//20://NG流道伺服上电
//	fbNGStepMotor.xPowerInit:=TRUE;
//	IF     fbNGStepMotor.xPowerOn THEN
//		station.iStepInit :=30;
//	END_IF
30://判断电动夹爪是否可以初始化
	IF    (tsModuleProcess[4].xProcessStarted AND  NOT tsModuleProcess[4].xProcessCompleted) OR
		  (tsModuleProcess[5].xProcessStarted AND  NOT tsModuleProcess[5].xProcessCompleted)  OR test THEN
			station.iStepInit :=50;(*电动夹爪不能初始h化*)
	ELSE
			station.iStepInit :=40;
	END_IF
40://大寰夹爪初始化
		fbClamp.stOper.xInitControl:=TRUE ;	
		 IF fbClamp.xDone  THEN 
				fbClamp.xExecute :=FALSE;
				station.iStepInit:=45;
		 END_IF	
45://大寰夹爪张开
			fbClamp.stOper.aReleaseControl[1]:=TRUE ;
				IF fbClamp.xDone  THEN 
					fbClamp.xExecute :=FALSE ;
					station.iStepInit:= 50;
				END_IF		
50:  //机械手初始化
		stToRobot1.iMoveMode := CmdRobot1.Cmd_GoHome ;//切换到回原点
		fbRobot.xInitExte := TRUE ;	
		station.iStepInit:=60;		
60:
		IF fbRobot.xInitFinish THEN 
			fbRobot.xInitExte := FALSE ;	
			station.iStepInit:=65;		
		END_IF		
65:
			//stToRobot1.iMoveMode := CmdRobot1.Cmd_GoHome ;
			station.iStepInit:=70;	
70://机械手初始化	
		IF  stFromRobot1.xStepRunning THEN
		 		station.iStepInit:=80;	
				stToRobot1.iMoveMode := CmdRobot1.noCmd ;
		END_IF
80://运行初始化子程序
		stToRobot1.xStepRunPermit := TRUE ;
	 IF stFromRobot1.xStepRunDone  THEN
		stToRobot1.xStepRunPermit := FALSE ;
   		station.iStepInit:=90;	
	 END_IF
90://机械手初始化并检测机械手初始化完成
	 IF  stFromRobot1.xHomePosReached THEN
        station.iStepInit:=999;	
	 END_IF	

999://初始化完成	
	station.iStepInit:=0;
	station.xInitDone:=TRUE;  
END_CASE
END_IF
END_ACTION

ACTION General:
EstopR_TRIG(CLK:= NOT  fbMachine[1].xEStop , Q=> );
IF  EstopR_TRIG.Q THEN 
		xS07MainlineRunPermit:=FALSE;
END_IF
MachineInitR_TRIG(CLK:=fbMachine[1].xIniting , Q=> );
IF MachineInitR_TRIG.Q THEN
		bRobCounter :=0;
END_IF
END_ACTION

ACTION ILC:

//---------------------------------------------------工站可执行-------------------------------------------------------
station.xCanRun :=TRUE ;

//---------------------------------------------------伺服动作条件-------------------------------------------
fbNGStepMotor.xRunILC := TRUE;
fbNGStepMotor.xMoveILC[1] :=TRUE;
//大寰夹爪
fbClamp.xDeviceRunning:=station.xSingleRunning OR   station.xIniting OR   station.xRunning ;
END_ACTION

ACTION TipAuto:

//------------------------------------------------AutoTip Cylinder--------------------------------

//------------------------------------------------AutoTip Servo--------------------------------
//**************************************
//FOR i:= 1 TO 5 BY 1 DO 
//	IF fbNGStepMotor.xMoveAuto[i] THEN
//		fbNGStepMotor.iPosNumber := i ;
//	END_IF
//	
//END_FOR
//
//
//IF  fbMachine[1].xAutoMode AND NOT fbMachine[1].xRunning AND  arTonDelay[10].Q   THEN
//		IF	fbNGStepMotor.iPosNumber=1 	AND NOT fbNGStepMotor.xMoveInPos[1] THEN 	station.adwAutoTip[1].10:=TRUE	;	END_IF//轴伺服自动时位置不在位置1
//		IF	fbNGStepMotor.iPosNumber=2	AND NOT fbNGStepMotor.xMoveInPos[2]	THEN 	station.adwAutoTip[1].11:=TRUE	;	END_IF//轴伺服自动时位置不在位置2
//		IF	fbNGStepMotor.iPosNumber=3	AND NOT fbNGStepMotor.xMoveInPos[3]	THEN 	station.adwAutoTip[1].12:=TRUE	;	END_IF//轴伺服自动时位置不在位置3
//		IF	fbNGStepMotor.iPosNumber=4	AND NOT fbNGStepMotor.xMoveInPos[4]	THEN 	station.adwAutoTip[1].13:=TRUE	;	END_IF//轴伺服自动时位置不在位置4
//		IF	fbNGStepMotor.iPosNumber=5	AND NOT fbNGStepMotor.xMoveInPos[5]	THEN 	station.adwAutoTip[1].14:=TRUE	;	END_IF//轴伺服自动时位置不在位置5
//END_IF
//
END_ACTION

ACTION TipManual:
//--------------------------------------------ManualTip------------------------------------------------------

//-------------------------------------------气缸提示---------------------------------------------------------




/////////////////////////////////////////////////////////////////////////////////////////////////////////////////
END_ACTION

ACTION Z_Output:
(*
CASE  bRobotStep  OF
 0:
 		IF   xRobotStartTryRun  THEN
		 		 bRobotStep:=bRobotStep +1;
		END_IF
1:  //机械手初始化
		fbRobot.xInitExte := TRUE ;
		 bRobotStep:=bRobotStep +1;
2:
		IF fbRobot.xInitFinish THEN 
			fbRobot.xInitExte := FALSE ;	
			 bRobotStep:=bRobotStep +1;
		END_IF		
3://机械手初始化	
		stToRobot1.iMoveMode := CmdRobot1.Cmd_GoHome ;
		IF  stFromRobot1.xStepRunning THEN
		 		 bRobotStep:=bRobotStep +1;
				stToRobot1.iMoveMode := CmdRobot1.noCmd ;
		END_IF
4://运行初始化子程序
		stToRobot1.xStepRunPermit := TRUE ;
	 IF stFromRobot1.xStepRunDone  THEN
		stToRobot1.xStepRunPermit := FALSE ;
   	 bRobotStep:=bRobotStep +1;
	 END_IF
5://机械手初始化并检测机械手初始化完成
	 IF  stFromRobot1.xHomePosReached THEN
       bRobotStep:=bRobotStep +1;
	 END_IF	
6://机械手选择取料程序	
			stToRobot1.iMoveMode := CmdRobot1.Cmd_TakePart ;//切换程序
			IF    stFromRobot1.xStepRunning  THEN
			 			stToRobot1.iMoveMode := CmdRobot1.noCmd ;
			 			 bRobotStep:=bRobotStep +1;
			END_IF
7://取料子程序运行
			stToRobot1.xStepRunPermit := TRUE ;
			IF stFromRobot1.xStepRunDone THEN
					stToRobot1.xStepRunPermit := FALSE ;
					 bRobotStep:=bRobotStep +1;
	 		END_IF
8:	//机械手允许去取料位
				 	stToRobot1.xPickPos1Premit :=TRUE;
						IF stFromRobot1.xPickPos1Reached THEN 
							 stToRobot1.xPickPos1Premit := FALSE ;
							 	 bRobotStep:=bRobotStep +1;
						END_IF
9://夹取完成,机械手回中转位
				stToRobot1.xClampPartDone:=TRUE;
			IF   stFromRobot1.xPickTransferPosReached THEN
					 bRobotStep:=bRobotStep +1;
			END_IF
10:
			stToRobot1.iMoveMode := CmdRobot1.Cmd_PutPart ;//切换程序
			IF    stFromRobot1.xStepRunning  THEN
			 			stToRobot1.iMoveMode := CmdRobot1.noCmd ;
			 		 bRobotStep:=bRobotStep +1;
			END_IF
11://放料子程序运行
			stToRobot1.xStepRunPermit := TRUE ;
			IF stFromRobot1.xStepRunDone THEN
					stToRobot1.xStepRunPermit := FALSE ;
					 bRobotStep:=bRobotStep +1;
	 		END_IF
12:	//机械手开始放料
			stToRobot1.xPutPos1Premit:=TRUE;(*卡片1位置 *)
			IF stFromRobot1.xPutPos1Reached THEN 
				 stToRobot1.xPutPos1Premit := FALSE ;
				 bRobotStep:=bRobotStep +1;
			END_IF
13://机械手回中转位置
			stToRobot1.xReleasePartDone:=TRUE;
			IF stFromRobot1.xPickTransferPosReached THEN
					bRobotStep:=0;
	 		END_IF	
END_CASE
*)
END_ACTION

END_PROGRAM

// ---- POUs/003_FB/0013_RGI_14_new/不带旋转的电动夹爪/FB_RGI_14_Modbus.TcPOU
{attribute 'tc_no_symbol'}
FUNCTION_BLOCK FB_RGI_14_Modbus
VAR_INPUT
	xExecute: BOOL;
	xAbort: BOOL;
	xPowerHmi: BOOL := TRUE;
	////上电信号，反转型
	xResetRequest: BOOL;
	///[ms],1 => no invocation time limit
	dwTimeLimit: DWORD := 1;
	///[ms],0 => no executing time limit 
	dwTimeOut: DWORD;
	///系统参数
	stPara: ST_RGI_14_Sys_Para;
	///0:mannal 1:auto
	xAutoMode: BOOL;
	///初始化过程中	
	xIniting: BOOL;
	///参数设置
	stPosPara: ST_RGI_PosPara;
	///流程运行过程中
	xDeviceRunning: BOOL;
	///手动自动操作
	stOper: ST_RGI_Opera;
END_VAR
VAR_OUTPUT
	///完成条件满足
	xDone: BOOL;
	///动作正在执行
	xBusy: BOOL;
	///指令被打断
	xAborted: BOOL;
	///错误条件满足
	xError: BOOL;
	///错误码
	eErrorID: RGI_14_ERROR;
	///eMobbusErrorID: MODBUS_ERROR;//modubs 报警信息
	xRdyCmd: BOOL;
	xRefOk: BOOL;
	eClampActCmd: RGI_14_CMD;
	///0：运动中，1：到达位置；2：夹住物体；3：物体掉落	
	iClampStatus: INT;
	///夹爪夹空
	xGripClampEmpty: BOOL;
	///掉落发生
	xDropOccur: BOOL;
	///关盖失败
	xClosecoverFailure: BOOL;
	///开盖失败
	xOpencoverFailure: BOOL;
	sHmiError: STRING;
	stRGIStates: ST_RGI_HMIStates;
	eCommErrorID: BYTE;
	eOperErrorID: DWORD;
END_VAR
VAR_IN_OUT
	st_IOData: ST_RGI_14_IOData;
END_VAR
VAR
	{attribute 'tc_no_symbol'}
	_xDone: BOOL;
	{attribute 'tc_no_symbol'}
	eCmd: RGI_14_CMD;
	{attribute 'tc_no_symbol'}
	///目标力值设置
	iTorqueSet: INT := 50;
	{attribute 'tc_no_symbol'}
	///运行速度设置
	iSpeedSet: INT := 50;
	{attribute 'tc_no_symbol'}
	///位置和速度设置值	
	iPosAngleSet: INT := 500;
	{attribute 'tc_no_symbol'}
	eState: STATE;
	{attribute 'tc_no_symbol'}
	xFirstInvocation: BOOL := TRUE;
	{attribute 'tc_no_symbol'}
	xTimeOut: BOOL;
	{attribute 'tc_no_symbol'}
	tOperationTimer: TON;
	{attribute 'tc_no_symbol'}
	_tonTimeout: TON;
	{attribute 'tc_no_symbol'}
	_tonCmdTimeout: TON;
	{attribute 'tc_no_symbol'}
	_tonPulse: TON;
	{attribute 'tc_no_symbol'}
	_tonDelay: TON;
	{attribute 'tc_no_symbol'}
	_tonConnectDelay: TON;
	{attribute 'tc_no_symbol'}
	_tonConnectTimeout: TON;
	{attribute 'tc_no_symbol'}
	/// detect rising edge of command execution 
	_diCmdState: DINT;
	{attribute 'tc_no_symbol'}
	i: INT;
	{attribute 'tc_no_symbol'}
	ii: INT;
	{attribute 'tc_no_symbol'}
	_idx: INT;
	{attribute 'tc_no_symbol'}
	_xConnectError: BOOL;
	{attribute 'tc_no_symbol'}
	_fResetCheck: F_TRIG;
	{attribute 'tc_no_symbol'}
	_iRotateAngleLTemp: INT;
	{attribute 'tc_no_symbol'}
	_iRotateAngleHTemp: INT;
	{attribute 'tc_no_symbol'}
	_iRotateAngleTotalTemp: DINT;
	{attribute 'tc_no_symbol'}
	_iRotateAngleCurrentTemp: DINT;
	{attribute 'tc_no_symbol'}
	_xRotateFinish: BOOL;
	{attribute 'tc_no_symbol'}
	_iConnectState: INT := 0;
	{attribute 'tc_no_symbol'}
	_connectTon: TON;
	{attribute 'tc_no_symbol'}
	_rManual: R_TRIG;
	{attribute 'tc_no_symbol'}
	_fManual: F_TRIG;
	{attribute 'tc_no_symbol'}
	_xModeChange: BOOL;
	{attribute 'tc_no_symbol'}
	///上电是默认读取模式的
	_xReadStatus: BOOL := TRUE;
	{attribute 'tc_no_symbol'}
	_iCount: INT := 0;
	{attribute 'tc_no_symbol'}
	_iAbortState: INT := 0;
	{attribute 'tc_no_symbol'}
	_fPowerOn :F_TRIG;
  {attribute 'tc_no_symbol'}
	_rHMIControl: R_TRIG;
	{attribute 'tc_no_symbol'}
	_iNGCount: INT;
	{attribute 'tc_no_symbol'}
	///4:控制反馈数据，5:状态反馈数据
	_aRead_VAR: ARRAY[4..5] OF FB_MBReadRegs;
	{attribute 'tc_no_symbol'}
	///0:初始化控制；1:夹紧控制；2:旋转绝对控制；3:旋转相对控制
	_aWtirt_VAR: ARRAY[0..3] OF FB_MBWriteRegs;
	{attribute 'tc_no_symbol'}
	///0:初始化控制；1:夹紧控制；2:旋转绝对控制；3:旋转相对控制；4:控制反馈数据，5:状态反馈数据	
	_aEnableSignal: ARRAY[0..5] OF BOOL;
	{attribute 'tc_no_symbol'}
	///反馈数据	
	_aFeedbackData: ARRAY[4..5, 0..11] OF INT;
	{attribute 'tc_no_symbol'}
	///控制参数	
	_aControlData: ARRAY[0..3, 0..3] OF INT;
	{attribute 'tc_no_symbol'}
	_iChannelIndex: INT;
	{attribute 'tc_no_symbol'}
	_xConnect_ERROR: BOOL;
	{attribute 'tc_no_symbol'}
	iCMDNGIndex: INT;
	{attribute 'tc_no_symbol'}
	_xBusy: BOOL;
	{attribute 'tc_no_symbol'}
	///发送状态标志位
	_iSendReceiveState: INT := 0;
	{attribute 'tc_no_symbol'}
	_tonDelay1: TON;
	{attribute 'tc_no_symbol'}
	_tonDelay2: TON;
	{attribute 'tc_no_symbol'}
	_iComNGCount: INT;
	{attribute 'tc_no_symbol'}
	///初始化指令触发
	_rHMIInit: R_TRIG;
	{attribute 'tc_no_symbol'}
	///初始化指令触发
	_rInit: R_TRIG;
	{attribute 'tc_no_symbol'}
	///夹紧轴指令触发
	_rHMIClamp: ARRAY[1..10] OF R_TRIG;
	{attribute 'tc_no_symbol'}
	///夹紧轴指令触发
	_rHMIRelease: ARRAY[1..10] OF R_TRIG;
	{attribute 'tc_no_symbol'}
	///夹紧轴指令触发
	_rClamp: ARRAY[1..10] OF R_TRIG;
	{attribute 'tc_no_symbol'}
	///夹紧轴指令触发
	_rRelease: ARRAY[1..10] OF R_TRIG;
	{attribute 'tc_no_symbol'}
	///旋转轴指令触发	
	_rHMIRotateClamp: ARRAY[1..10] OF R_TRIG;
	{attribute 'tc_no_symbol'}
	///旋转轴指令触发	
	_rHMIRotateClampRef: ARRAY[1..10] OF R_TRIG;
	{attribute 'tc_no_symbol'}
	///旋转轴指令触发	
	_rHMIRotateRelease: ARRAY[1..10] OF R_TRIG;
	{attribute 'tc_no_symbol'}
	///旋转轴指令触发	
	_rHMIRotateReleaseRef: ARRAY[1..10] OF R_TRIG;
	{attribute 'tc_no_symbol'}
	///旋转轴指令触发	
	_rRotateClamp: ARRAY[1..10] OF R_TRIG;
	{attribute 'tc_no_symbol'}
	///旋转轴指令触发	
	_rRotateRelease: ARRAY[1..10] OF R_TRIG;
	{attribute 'tc_no_symbol'}
	///旋转轴指令触发	
	_rRotateClampRef: ARRAY[1..10] OF R_TRIG;
	{attribute 'tc_no_symbol'}
	///旋转轴指令触发	
	_rRotateReleaseRef: ARRAY[1..10] OF R_TRIG;
	{attribute 'tc_no_symbol'}
	_Angle_rec: INT;
	{attribute 'tc_no_symbol'}
	///是否有手动操作，是否有自动操作
	_xHMIOpe: BOOL;
	{attribute 'tc_no_symbol'}
	///是否有手动操作，是否有自动操作
	_xAutoOpe: BOOL;
END_VAR
VAR_TEMP
	{attribute 'tc_no_symbol'}
	xAgain: BOOL;
END_VAR

xAgain:=0;
ACTMap();//数据映射
ConnectAction();//触发通信连接功能连接
_fResetCheck(CLK:=xResetRequest OR stOper.xHMIReset);//reset
IF eState<>STATE.DORMANT
THEN
	_rHMIInit(CLK:=FALSE) ;
	_rInit(CLK:=FALSE) ;
	 FOR ii :=1 TO 10 DO
		 _rHMIClamp[ii](CLK:=FALSE);
		 _rHMIRelease[ii](CLK:=FALSE);
		 _rClamp[ii](CLK:=FALSE);
		 _rRelease[ii](CLK:=FALSE);
		 _rHMIRotateClamp[ii](CLK:=FALSE);
		 _rHMIRotateRelease[ii](CLK:=FALSE);
		 _rRotateClamp[ii](CLK:=FALSE);
		 _rRotateRelease[ii](CLK:=FALSE);
		 _rRotateClampRef[ii](CLK:=FALSE);
		 _rRotateReleaseRef[ii](CLK:=FALSE);
		 _rHMIRotateClampRef[ii](CLK:=FALSE);
		 _rHMIRotateReleaseRef[ii](CLK:=FALSE);		 
	 END_FOR
END_IF
REPEAT
	CASE eState OF
		STATE.DORMANT:
				HandleDormantState(xAgain=> xAgain);
		STATE.EXECUTING:
				HandleExecutingState(xAgain=> xAgain);
		STATE.DONE:
				HandleDoneState(xAgain=> xAgain);
		STATE.INERROR:
				HandleErrorState(xAgain=> xAgain);
		STATE.ABORTING:
				HandleAbortingState(xAgain=> xAgain);
		STATE.ABORTED:
				HandleAbortedState(xAgain=> xAgain);
		STATE.RESETING:
				HandleResettingState(xAgain=> xAgain);
	END_CASE
UNTIL (xAgain=0)
END_REPEAT

//报错信息提示	
CASE eErrorID OF
	RGI_14_ERROR.NO_ERROR:
		sHmiError:='NO_ERROR';	
  RGI_14_ERROR.FLT_PARA:
		sHmiError:='FLT_PARA';	
  RGI_14_ERROR.FLT_CONNECT:
		sHmiError:='FLT_CONNECT';	
  RGI_14_ERROR.FLT_RDYCMD:
		sHmiError:='FLT_RDYCMD';	
	RGI_14_ERROR.FLT_DEVICE_ERROR:
		sHmiError:='FLT_DEVICE_ERROR';	
	RGI_14_ERROR.FLT_POWERON:
		sHmiError:='FLT_POWERON';	
  RGI_14_ERROR.FLT_CLAMP_TIMEOUT:
		sHmiError:='FLT_CLAMP_TIMEOUT';	
  RGI_14_ERROR.FLT_ROTATE_TIMEOUT:
		sHmiError:='FLT_ROTATE_TIMEOUT';	
  RGI_14_ERROR.FLT_ORG_TIMEOUT:
		sHmiError:='FLT_ORG_TIMEOUT';	
	RGI_14_ERROR.FLT_CLAMPCMD_TIMEOUT:
		sHmiError:='FLT_CLAMPCMD_TIMEOUT';	
  RGI_14_ERROR.FLT_ROTATECMDABS_TIMEOUT:
		sHmiError:='FLT_ROTATECMDABS_TIMEOUT';
  RGI_14_ERROR.FLT_ROTATECMDREF_TIMEOUT:
		sHmiError:='FLT_ROTATECMDREF_TIMEOUT';			
  RGI_14_ERROR.FLT_ORGCMD_TIMEOUT:
		sHmiError:='FLT_ORGCMD_TIMEOUT';	
	RGI_14_ERROR.FLT_CLAMP_DROP:
		sHmiError:='FLT_CLAMP_DROP';	  
  RGI_14_ERROR.FLT_xRefOk:
		sHmiError:='FLT_xRefOk';	
	RGI_14_ERROR.FLT_CLAMP_PARA:
		sHmiError:='FLT_CLAMP_PARA';		
	RGI_14_ERROR.FLT_ClAMP_RELEASEFAIL:
		sHmiError:='FLT_ClAMP_RELEASEFAIL';	
  RGI_14_ERROR.FLT_ClAMP_CLAMPFAIL:
		sHmiError:='FLT_ClAMP_CLAMPFAIL';	
	RGI_14_ERROR.FLT_ROTATE_CLAMPFAIL:
		sHmiError:='FLT_ROTATE_CLAMPFAIL';	
	RGI_14_ERROR.FLT_ROTATE_RELEASEFAIL:
		sHmiError:='FLT_ROTATE_RELEASEFAIL';		
END_CASE

//检测是否有手动操作
_xHMIOpe := stOper.xHMInitButton;
FOR i := 1 TO 10 BY 1
DO
	_xHMIOpe := _xHMIOpe OR stOper.aHMIClampButton[i] OR stOper.aHMIReleaseButton[i] OR stOper.aHMIRotateClampButton[i] OR stOper.aHMIRotateClampRefButton[i] 
							OR stOper.aHMIRotateReleaseButton[i] OR stOper.aHMIRotateReleaseRefButton[i];
END_FOR

//检测是否有自动操作指令
_xAutoOpe := stOper.xInitControl;
FOR i := 1 TO 10 BY 1
DO
	_xAutoOpe := _xAutoOpe OR stOper.aClampControl[i] OR stOper.aReleaseControl[i] OR stOper.aRotateClampControl[i] OR stOper.aRotateClampRefControl[i] 
							OR stOper.aRotateReleaseControl[i] OR stOper.aRotateReleaseRefControl[i];
END_FOR

///{attribute 'tc_no_symbol'}
METHOD PROTECTED AbortAction
VAR_OUTPUT
	xComplete: BOOL;
	eErrorID: RGI_14_ERROR;
END_VAR
(*
* Cleaning
* => abort all running operation
* => if an NBS.ERROR codition is reached, set eErrorID to a Value rather then NBS.RGI_14_ERROR.NO_ERROR 
*)
CASE _iAbortState OF 
	0://复位所以的控制信号

	ELSE
		;	
END_CASE
END_METHOD

ACTION ACTCheckRotateFinish:
(******************************检测旋转是否完成*************************************)
_xRotateFinish := FALSE;
IF eCmd = RGI_14_CMD.Cmd_RotateAbsClamp OR eCmd = RGI_14_CMD.Cmd_RotateAbsRelease //绝对旋转模式
THEN
	//检测是否已经处于目标位置
	IF iPosAngleSet = st_IOData.I_RotateAngleL
	THEN
		_xRotateFinish := TRUE;
	END_IF	
END_IF
IF eCmd = RGI_14_CMD.Cmd_RoratRelClamp OR eCmd = RGI_14_CMD.Cmd_RoratRelRelease//增量旋转模式
THEN	
	//使用计算公式来进行预测是否已经到目标位置
	_iRotateAngleTotalTemp := _iRotateAngleHTemp * 32768 + _iRotateAngleLTemp + iPosAngleSet;
	_iRotateAngleCurrentTemp := st_IOData.I_RotateAngleH * 32768 + st_IOData.I_RotateAngleL;
	IF _iRotateAngleTotalTemp = _iRotateAngleCurrentTemp
	THEN
		_xRotateFinish := TRUE;
	END_IF
END_IF
END_ACTION

ACTION ACTMap:
//进行数据映射的前提条件是外部所配置的参数是没有问题的
IF stPara.strSlaveIP <> '' 
THEN
	//夹爪设置反馈
	st_IOData.i_Init			:=_aFeedbackData[4,0];
	st_IOData.i_ClampForceSet	:=_aFeedbackData[4,1];
	
	st_IOData.i_ClampPosSet		:=_aFeedbackData[4,3];	
	st_IOData.i_ClampSpeedSet	:=_aFeedbackData[4,4];
	st_IOData.i_RotateAngleLSet	:=_aFeedbackData[4,5];
	st_IOData.i_RotateAngleHSet	:=_aFeedbackData[4,6];
	st_IOData.i_RotateSpeedSet	:=_aFeedbackData[4,7];
	st_IOData.i_RotateForseSet	:=_aFeedbackData[4,8];
	st_IOData.i_RotateRelAngle	:=_aFeedbackData[4,9];
	
	//夹爪状态反馈
	st_IOData.I_ClampInit := _aFeedbackData[5,0];
	st_IOData.I_ClampState := _aFeedbackData[5,1];
	st_IOData.I_CurrentPos := _aFeedbackData[5,2];
	st_IOData.I_DeviceERRORState := _aFeedbackData[5,5];
	st_IOData.I_RotateAngleL := _aFeedbackData[5,8];
	st_IOData.I_RotateAngleH := _aFeedbackData[5,9];
	st_IOData.I_RotateInit := _aFeedbackData[5,10];
	st_IOData.I_RotateState := _aFeedbackData[5,11];			
	//夹爪状态
	iClampStatus := st_IOData.I_ClampState ;
	
	//进行输出数据刷新(外面一定要用保持性的数据来定义)
	_aControlData[0,0] := st_IOData.O_Init;//同时初始化夹紧轴和旋转轴
	_aControlData[1,0] := st_IOData.O_ClampForceSet;//夹紧力值设计
	_aControlData[1,2] := st_IOData.O_ClampPosSet;//夹紧位置设置
	_aControlData[1,3] := st_IOData.O_ClampSpeedSet;//夹紧速度设置
	//旋转绝对定位
	IF eCmd = RGI_14_CMD.Cmd_RotateAbsClamp OR eCmd = RGI_14_CMD.Cmd_RotateAbsRelease
	THEN
		_aControlData[2,0]	:= st_IOData.O_RotateAngleLSet;//绝对旋转角度设置1
		_aControlData[2,1] := st_IOData.O_RotateAngleHSet;//绝对旋转角度设置2	
		_aControlData[2,2] := st_IOData.O_RotateSpeedSet;//旋转速度设计
		_aControlData[2,3] := st_IOData.O_RotateForseSet;//旋转力值设计		
	END_IF
	//旋转相对定位
	IF eCmd = RGI_14_CMD.Cmd_RoratRelClamp OR eCmd = RGI_14_CMD.Cmd_RoratRelRelease
	THEN
		_aControlData[3,0] := st_IOData.O_RotateSpeedSet;//旋转速度设计
		_aControlData[3,1] := st_IOData.O_RotateForseSet;//旋转力值设计
		_aControlData[3,2] := st_IOData.O_RotateRelAngle;//旋转相对角度设计
	END_IF
	
END_IF

(****************************夹紧轴状态读取(此时一定是模块连接上的，此时刷新周期不要太短，兼容效率***************************)
_tonPulse(IN:=NOT _tonPulse.Q , PT:=T#200MS);//产生100ms的脉冲信号
IF _xReadStatus  //一定要处于通信正常状态
THEN
	_aRead_VAR[5].bExecute := _tonPulse.Q;//保证通信不断
END_IF

xRdyCmd := xPowerHmi AND(( eState = STATE.DORMANT ) OR (NOT xAutoMode AND _xAutoOpe AND eState = STATE.DONE ));//rdy显示变化;
_rInit(CLK:= xIniting);//检测是否是初始化中，如果是的去切换模式
IF _rInit.Q
THEN
 eState := STATE.RESETING;
END_IF 
//检测是否有模式变化
_fManual(CLK:=xAutoMode);
_rManual(CLK:=xAutoMode);
IF eState <> STATE.DORMANT//只有在运行的时候，才会检测是否有模式切换发生
THEN
	IF _fManual.Q OR _rManual.Q
	THEN
		_xModeChange := TRUE;
	END_IF
END_IF

(****************************电源控制********************************************)

_fPowerOn(CLK:= xPowerHmi);//驱动器断电的时候需要将初始化完成信号给清除掉
IF _fPowerOn.Q
THEN
	xRefOk := FALSE;//断电再上电之后需要重新初始化
END_IF

(*****************************夹爪状态显示*****************************)
xDone := _xDone AND xExecute;//判断是否处于当前流程的Done状态
xDropOccur :=( eClampActCmd = RGI_14_CMD.Cmd_Clamp ) AND ( st_IOData.I_ClampState = 3 );
xGripClampEmpty := xError AND eErrorID = RGI_14_ERROR.FLT_ClAMP_CLAMPFAIL AND xExecute;//关盖失败判定
xClosecoverFailure := xError AND eErrorID = RGI_14_ERROR.FLT_ROTATE_CLAMPFAIL AND xExecute;//关盖失败判定
xOpencoverFailure := xError AND eErrorID = RGI_14_ERROR.FLT_ROTATE_RELEASEFAIL AND xExecute;//开盖失败评定

(*****************************触摸屏状态显示*****************************)
stRGIStates.xDone:=xDone;
stRGIStates.xBusy:=xBusy;
stRGIStates.xRefOk:=xRefOk;
stRGIStates.xRdyCmd:=xRdyCmd;
stRGIStates.eErrorID:=eErrorID;
stRGIStates.sHmiError:=sHmiError;
stRGIStates.iClampStatus:=iClampStatus;
stRGIStates.xClosecoverFailure:=xClosecoverFailure;
stRGIStates.xGripClampEmpty:=xGripClampEmpty;
stRGIStates.xOpencoverFailure:=xOpencoverFailure;
stRGIStates.xGripClampEmpty:=xGripClampEmpty;
stRGIStates.xError:=xError;
END_ACTION

METHOD PROTECTED CmdClampAction
VAR_OUTPUT
	xComplete: BOOL;
END_VAR
// return the real actual fault number
IF eErrorID <> RGI_14_ERROR.NO_ERROR
THEN
  RETURN;  
END_IF
  
IF NOT xRefOk THEN
	eErrorID := RGI_14_ERROR.FLT_xRefOk;
	RETURN;
END_IF

IF iPosAngleSet < 0 OR iPosAngleSet > 1000//夹紧参数错误
THEN
	eErrorID := RGI_14_ERROR.FLT_CLAMP_PARA;
	RETURN;
END_IF

CASE _diCmdState OF
	0://判断对应指令，是否已经处于完成状态，防止出现重复触发情况
		_tonDelay(IN:= FALSE);
		IF NOT _aRead_VAR[5].bExecute THEN		
			_diCmdState := _diCmdState + 1;
		END_IF	
		
	1://传送力值和速度参数
		_tonDelay(IN:= TRUE,pt:=T#20MS);
		st_IOData.O_ClampForceSet	:= iTorqueSet;
		st_IOData.O_ClampSpeedSet	:= iSpeedSet;	
		st_IOData.O_ClampPosSet 	:= iPosAngleSet;	
		IF _tonDelay.Q 
		THEN
			//复位定时器
				_tonDelay(IN:=FALSE);
				_tonCmdTimeout(in:=FALSE);
				_tonTimeout(in:=FALSE);	
			 _aEnableSignal[1]:=TRUE;	
			 _diCmdState := _diCmdState+1;
	 END_IF				
		
	2://等待反应，设置读取参数
		_tonDelay(IN:= NOT _aEnableSignal[1],PT:=T#300MS);//此时电动夹爪一定已经响应
		IF _tonDelay.Q//
		THEN		
			_diCmdState := _diCmdState +1;			
		END_IF	
		
		IF _iSendReceiveState = 999
		THEN
			iCMDNGIndex := 1;
			eErrorID := RGI_14_ERROR.FLT_CLAMPCMD_TIMEOUT;		
			_diCmdState := 999;
		END_IF	
		
	3://读取数据
		_tonCmdTimeout(in:=FALSE);
		_tonDelay(IN:=FALSE);	
		_tonTimeout(in:=TRUE,pt:=T#10S);//设置超时时间 
		_aEnableSignal[5] := TRUE;//触发读取反馈数据	
		_diCmdState := _diCmdState +1; 
	
	4://等待运行完成
		_tonTimeout(in:=TRUE,pt:=T#10S); 
		_tonCmdTimeout(IN:= TRUE,pt:=T#2S);				
		IF NOT _aEnableSignal[5] //等待读取数据完成
		THEN	
			_tonDelay(IN:= TRUE,pt:=T#40MS);//设置刷新周期
			IF _tonDelay.Q
			THEN
				_diCmdState := 3;//回到上一步重新进行状态刷新
			END_IF
			
			IF (st_IOData.I_ClampState = 1 OR stOper.xTestMode )AND st_IOData.O_ClampPosSet = st_IOData.I_CurrentPos AND //松开位置成功
			   eCmd = RGI_14_CMD.Cmd_Release	//松开指令
			THEN			
				_tonCmdTimeout(in:=FALSE);
				_tonTimeout(in:=FALSE);  
				_diCmdState := 100;
				xComplete := TRUE;
			END_IF		
			IF (st_IOData.I_ClampState = 2 OR stOper.xTestMode) AND//夹住物体
				 eCmd = RGI_14_CMD.Cmd_Clamp	//夹紧指令
			THEN			
				_tonTimeout(in:=FALSE);  
				_diCmdState := 100;
				xComplete := TRUE;
			END_IF			
		//非测试模式才启动检测
		IF NOT stOper.xTestMode THEN	
			IF st_IOData.I_ClampState = 2 AND //松开位置的时候，没有松开到位置，松开失败
				 eCmd = RGI_14_CMD.Cmd_Release	//松开指令
			THEN	
				_iNGCount := _iNGCount + 1;		
				IF _iNGCount <= 3
				THEN
					_tonDelay(IN:=FALSE);
					_diCmdState := _diCmdState + 1;
				ELSE
					_tonTimeout(in:=FALSE);  
					eErrorID := RGI_14_ERROR.FLT_ClAMP_RELEASEFAIL;		
					_diCmdState := 999;
				END_IF				
			END_IF		
			IF st_IOData.I_ClampState = 1 AND st_IOData.O_ClampPosSet = st_IOData.I_CurrentPos AND//没有夹住物体，到位置，判定夹持失败
				 eCmd = RGI_14_CMD.Cmd_Clamp	//夹紧指令
			THEN
				_iNGCount := _iNGCount + 1;		
				IF _iNGCount <= 3
				THEN
					_tonDelay(IN:=FALSE);
					_diCmdState := _diCmdState + 1;
				ELSE
					_tonCmdTimeout(in:=FALSE);
					_tonTimeout(in:=FALSE);  			
					eErrorID := RGI_14_ERROR.FLT_ClAMP_CLAMPFAIL;		
					_diCmdState := 999;
				END_IF
			END_IF		
		END_IF
	END_IF
	
	IF _iSendReceiveState = 999//旋转指令响应超时
	THEN
		iCMDNGIndex := 3;
		eErrorID := RGI_14_ERROR.FLT_CLAMPCMD_TIMEOUT;		
		_diCmdState := 999;
	END_IF		
	
	IF _tonTimeout.Q//旋转动作超时
	THEN
		_iNGCount := _iNGCount + 1;
		IF _iNGCount >= 2
		THEN
			eErrorID := RGI_14_ERROR.FLT_CLAMP_TIMEOUT;
			_diCmdState := 999;
		ELSE
			_aEnableSignal[5] := FALSE;
			_diCmdState := 0;
		END_IF
	END_IF
	
	5://报警再次确定
		_tonDelay(IN:= TRUE,pt:=T#50MS);
		IF _tonDelay.Q//做延时刷新
		THEN			
			_diCmdState :=3;
		END_IF
			
ELSE
	;	
END_CASE
END_METHOD

METHOD PROTECTED CmdRotateAction_ABS
VAR_OUTPUT
	xComplete: BOOL;
END_VAR
// return the real actual fault number
IF eErrorID <> RGI_14_ERROR.NO_ERROR
THEN
  RETURN;  
END_IF
  
IF NOT xRefOk THEN//设备没有原点报警
	eErrorID := RGI_14_ERROR.FLT_xRefOk;
	RETURN;
END_IF

CASE _diCmdState OF
	0://判断是否已经处于目标位置或者夹取完成状态，防止出现重复触发情况
		_tonDelay(IN:= FALSE);
		IF NOT _aRead_VAR[5].bExecute THEN		
			_diCmdState := _diCmdState + 1;
		END_IF		
		
	1://传送参数	
		_tonDelay(IN:= TRUE,PT:=T#20MS);//等待设备运行起来
		_iRotateAngleLTemp := st_IOData.I_RotateAngleL;
		_iRotateAngleHTemp := st_IOData.I_RotateAngleH;		
		st_IOData.O_RotateForseSet := iTorqueSet;
		st_IOData.O_RotateSpeedSet := iSpeedSet;
		st_IOData.O_RotateAngleLSet := iPosAngleSet;
		st_IOData.O_RotateRelAngle := 0;
		IF _tonDelay.Q 
		THEN
			//复位定时器
				_tonDelay(IN:=FALSE);
				_tonCmdTimeout(in:=FALSE);
				_tonTimeout(in:=FALSE);	
			 _aEnableSignal[2]:= TRUE;
			 _diCmdState := _diCmdState+1;
	 END_IF
	
		
	2://等待反应，设置读取参数
		_tonDelay(IN:= NOT _aEnableSignal[2],PT:=T#300MS);//此时电动夹爪一定已经响应
		IF _tonDelay.Q//
		THEN		
			_diCmdState := _diCmdState +1;			
		END_IF	
		
		IF _iSendReceiveState = 999
		THEN
			iCMDNGIndex := 1;
			eErrorID := RGI_14_ERROR.FLT_CLAMPCMD_TIMEOUT;		
			_diCmdState := 999;
		END_IF								
		
	3://读取数据
		_tonCmdTimeout(in:=FALSE);
		_tonDelay(IN:=FALSE);	
		_tonTimeout(in:=TRUE,pt:=T#10S);//设置超时时间 
		_aEnableSignal[5] := TRUE;//触发读取反馈数据	
		_diCmdState := _diCmdState +1; 		
				
	4://判定旋转结果
		_tonTimeout(in:=TRUE,pt:=T#10S); 
		_tonCmdTimeout(IN:= TRUE,pt:=T#2S);				
		IF NOT _aEnableSignal[5] //等待读取数据完成
		THEN	
			_tonDelay(IN:= TRUE,pt:=T#40MS);//设置刷新周期
			IF _tonDelay.Q
			THEN
				_diCmdState := 3;//回到上一步重新进行状态刷新
			END_IF
			
			IF ( ( st_IOData.I_RotateState = 1 AND _xRotateFinish ) OR st_IOData.I_RotateState = 3 OR stOper.xTestMode ) AND _xRotateFinish AND //旋转是否到位置,只有在松开瓶盖的时候会有这种操作
				 ( eCmd = RGI_14_CMD.Cmd_RotateAbsRelease)
			THEN			
				_tonTimeout(in:=FALSE);  
				_diCmdState := 100;
				xComplete := TRUE;
			END_IF		
			IF ( st_IOData.I_RotateState = 2 OR st_IOData.I_RotateState = 3 OR stOper.xTestMode ) AND //旋转夹瓶盖处理，只有出现堵转（达到设置力反馈）
				 ( eCmd = RGI_14_CMD.Cmd_RotateAbsClamp)
			THEN			
				_tonTimeout(in:=FALSE);  
				_diCmdState := 100;
				xComplete := TRUE;
			END_IF				
		//非测试模式才启动检测
			IF NOT stOper.xTestMode THEN
				IF ( st_IOData.I_RotateState = 1 AND _xRotateFinish ) AND //关盖打滑,直接到设置位置了
					 ( eCmd = RGI_14_CMD.Cmd_RotateAbsClamp )
				THEN
					_iNGCount := _iNGCount + 1;		
					IF _iNGCount <= 3//检测是否有正时报警发生
					THEN
						_tonDelay(IN:=FALSE);
						_diCmdState := _diCmdState + 1;
					ELSE
						eErrorID := RGI_14_ERROR.FLT_ROTATE_CLAMPFAIL;
						_diCmdState := 999;
					END_IF
				END_IF
				IF ( st_IOData.I_RotateState = 2 ) AND //开盖失败，直接堵转，开不开瓶盖
					 ( eCmd = RGI_14_CMD.Cmd_RotateAbsRelease)
				THEN	
					_tonDelay(IN:= st_IOData.I_RotateState = 2,pt:=T#500MS);//判断释放堵转
					IF _tonDelay.Q THEN
						_iNGCount := _iNGCount + 1;		
						IF _iNGCount <= 3//检测是否有正时报警发生
						THEN
							_tonDelay(IN:=FALSE);
							_diCmdState := _diCmdState + 1;
						ELSE
							eErrorID := RGI_14_ERROR.FLT_ROTATE_RELEASEFAIL;
							_tonDelay(IN:= FALSE,pt:=T#10MS);
							_diCmdState := 999;
						END_IF
					END_IF
				END_IF
			END_IF
		END_IF	
		IF _iSendReceiveState = 999//旋转指令响应超时
		THEN
			iCMDNGIndex := 3;
			eErrorID := RGI_14_ERROR.FLT_ROTATECMDABS_TIMEOUT;		
			_diCmdState := 999;
		END_IF		
		IF _tonTimeout.Q//回原点动作超时
		THEN
			eErrorID := RGI_14_ERROR.FLT_ROTATE_TIMEOUT;
			_diCmdState := 999;
		END_IF
		
	5://报警再次确定
		_tonDelay(IN:= TRUE,pt:=T#50MS);
		IF _tonDelay.Q//做延时刷新
		THEN			
			_diCmdState :=3;
		END_IF	

	
ELSE
	;	
END_CASE
ACTCheckRotateFinish();//调用计算是否到位置
END_METHOD

METHOD PROTECTED CmdRotateAction_Ref
VAR_OUTPUT
	xComplete: BOOL;
END_VAR
// return the real actual fault number
IF eErrorID <> RGI_14_ERROR.NO_ERROR
THEN
  RETURN;  
END_IF
  
IF NOT xRefOk THEN//设备没有原点报警
	eErrorID := RGI_14_ERROR.FLT_xRefOk;
	RETURN;
END_IF

CASE _diCmdState OF
	0://判断是否已经处于目标位置或者夹取完成状态，防止出现重复触发情况
		_tonDelay(IN:= FALSE);
		IF NOT _aRead_VAR[5].bExecute THEN		
			_diCmdState := _diCmdState + 1;
		END_IF	
		
	1://传送参数
	  	_tonDelay(IN:= TRUE,pt:=T#20MS);//保证执行的都是当次任务 			
			_iRotateAngleLTemp := st_IOData.I_RotateAngleL;
			_iRotateAngleHTemp := st_IOData.I_RotateAngleH;		
			st_IOData.O_RotateForseSet := iTorqueSet;
			st_IOData.O_RotateSpeedSet := iSpeedSet;
			st_IOData.O_RotateRelAngle := iPosAngleSet;				
			_Angle_rec:=st_IOData.I_RotateAngleL;//将当前夹爪旋转角度储存到缓存，用来判断机构是否动作
			IF _tonDelay.Q 
			THEN
			//复位定时器
				_tonDelay(IN:=FALSE);
				_tonCmdTimeout(in:=FALSE);
				_tonTimeout(in:=FALSE);	
			 _aEnableSignal[3]:= TRUE;
			 _diCmdState := _diCmdState+1;
			END_IF		


	2://等待反应，设置读取参数
		_tonDelay(IN:= NOT _aEnableSignal[3],PT:=T#300MS);//此时电动夹爪一定已经响应
		IF _tonDelay.Q//
		THEN		
			_diCmdState := _diCmdState +1;			
		END_IF	
		
		IF _iSendReceiveState = 999
		THEN
			iCMDNGIndex := 1;
			eErrorID := RGI_14_ERROR.FLT_ROTATECMDREF_TIMEOUT;		
			_diCmdState := 999;
		END_IF								
		
	3://读取数据
		_tonCmdTimeout(in:=FALSE);
		_tonDelay(IN:=FALSE);	
		_tonTimeout(in:=TRUE,pt:=T#10S);//设置超时时间 
		_aEnableSignal[5] := TRUE;//触发读取反馈数据	
		_diCmdState := _diCmdState +1; 
					
	4://判定旋转结果
		_tonTimeout(in:=TRUE,pt:=T#10S); 
		_tonCmdTimeout(IN:= TRUE,pt:=T#2S);				
		IF NOT _aEnableSignal[5] //等待读取数据完成
		THEN	
			_tonDelay(IN:= TRUE,pt:=T#40MS);//设置刷新周期
			IF _tonDelay.Q
			THEN
				_diCmdState := 3;//回到上一步重新进行状态刷新
			END_IF
			
			IF (  st_IOData.I_RotateState = 1 OR st_IOData.I_RotateState = 3 OR stOper.xTestMode ) AND //旋转是否到位置,只有在松开瓶盖的时候会有这种操作
				 ( eCmd = RGI_14_CMD.Cmd_RoratRelRelease )
			THEN			
				_tonTimeout(in:=FALSE);  
				_diCmdState := 100;
				xComplete := TRUE;
			END_IF		
			IF ( st_IOData.I_RotateState = 2 OR st_IOData.I_RotateState = 3 OR stOper.xTestMode ) AND //旋转夹瓶盖处理，只有出现堵转（达到设置力反馈）
				 ( eCmd = RGI_14_CMD.Cmd_RoratRelClamp )
			THEN			
				_tonTimeout(in:=FALSE);  
				_diCmdState := 100;
				xComplete := TRUE;
			END_IF				
			//非测试模式才启动检测
			IF NOT stOper.xTestMode THEN
				//关盖异常判断，关盖时直接旋转到位，没有遇到阻力判定为关盖失败
				IF ( st_IOData.I_RotateState = 1 ) AND //关盖打滑,直接到设置位置了,AND _Angle_rec+iPosAngleSet=st_IOData.I_RotateAngleL
					 ( eCmd = RGI_14_CMD.Cmd_RoratRelClamp )
				THEN
					_iNGCount := _iNGCount + 1;		
					IF _iNGCount <= 2//检测是否有正时报警发生
					THEN
						_tonDelay(IN:=FALSE);
						_diCmdState := 3;
					ELSE
						eErrorID := RGI_14_ERROR.FLT_ROTATE_CLAMPFAIL;
						_diCmdState := 999;
					END_IF
				END_IF
				//开盖异常判断
				IF ( st_IOData.I_RotateState = 2 ) AND //开盖失败，直接堵转，开不开瓶盖
					 ( eCmd = RGI_14_CMD.Cmd_RoratRelRelease )
				THEN	
					_tonDelay(IN:= st_IOData.I_RotateState = 2,pt:=T#500MS);//判断释放堵转
					IF _tonDelay.Q THEN
						_iNGCount := _iNGCount + 1;		
						IF _iNGCount <= 2//检测是否有正时报警发生
						THEN
							_tonDelay(IN:=FALSE);
							_diCmdState := 3;
						ELSE
							eErrorID := RGI_14_ERROR.FLT_ROTATE_RELEASEFAIL;
							_tonDelay(IN:= FALSE,pt:=T#10MS);
							_diCmdState := 999;
						END_IF
					END_IF
				END_IF
			END_IF
		END_IF	
		IF _iSendReceiveState = 999//旋转指令响应超时
		THEN
			iCMDNGIndex := 3;
			eErrorID := RGI_14_ERROR.FLT_ROTATECMDABS_TIMEOUT;		
			_diCmdState := 999;
		END_IF
		//超时判定
		IF _tonTimeout.Q//动作超时
		THEN
			eErrorID := RGI_14_ERROR.FLT_ROTATE_TIMEOUT;
			_diCmdState := 999;
		END_IF
		
	5://报警再次确定
		_tonDelay(IN:= TRUE,pt:=T#50MS);
		IF _tonDelay.Q//做延时刷新
		THEN			
			_diCmdState :=3;
		END_IF		
		
	ELSE
		;	
END_CASE
ACTCheckRotateFinish();//调用计算是否到位置
END_METHOD

ACTION ConnectAction:
	
(**********************************调用收发功能块**********************************)
//状态反馈功能调用
_aRead_VAR[4](
	sIPAddr:= stPara.strSlaveIP, 
	nTCPPort:= stPara.iSlavePort, 
	nUnitID:= stPara.bySlaveID, 
	nQuantity:= 10, 
	nMBAddr:=16#100 , 
	cbLength:= 20, 
	pDestAddr:=ADR(_aFeedbackData[4,0]));	
	
_aRead_VAR[5](
	sIPAddr:= stPara.strSlaveIP, 
	nTCPPort:= stPara.iSlavePort, 
	nUnitID:= stPara.bySlaveID, 
	nQuantity:= 12, 
	nMBAddr:=16#200 , 
	cbLength:= 24, 
	pDestAddr:=ADR(_aFeedbackData[5,0]));		
	
//指令控制部分
_aWtirt_VAR[0](
	sIPAddr:= stPara.strSlaveIP,
	nTCPPort:= stPara.iSlavePort, 
	nUnitID:= stPara.bySlaveID, 
	nQuantity:= 1, 
	nMBAddr:= 16#100, 
	cbLength:= 2, 
	pSrcAddr:= ADR(_aControlData[0,0]), 
	bExecute:= , 
	tTimeout:= T#1S, 
	bBusy=> , 
	bError=> , 
	nErrId=> );	
	
_aWtirt_VAR[1](
	sIPAddr:= stPara.strSlaveIP,
	nTCPPort:= stPara.iSlavePort, 
	nUnitID:= stPara.bySlaveID, 
	nQuantity:= 4, 
	nMBAddr:= 16#101, 
	cbLength:= 8, 
	pSrcAddr:= ADR(_aControlData[1,0]), 
	bExecute:= , 
	tTimeout:= T#1S, 
	bBusy=> , 
	bError=> , 
	nErrId=> );	
	
_aWtirt_VAR[2](
	sIPAddr:= stPara.strSlaveIP,
	nTCPPort:= stPara.iSlavePort, 
	nUnitID:= stPara.bySlaveID, 
	nQuantity:= 4, 
	nMBAddr:= 16#105, 
	cbLength:= 8, 
	pSrcAddr:= ADR(_aControlData[2,0]), 
	bExecute:= , 
	tTimeout:= T#1S, 
	bBusy=> , 
	bError=> , 
	nErrId=> );	
	
_aWtirt_VAR[3](
	sIPAddr:= stPara.strSlaveIP,
	nTCPPort:= stPara.iSlavePort, 
	nUnitID:= stPara.bySlaveID, 
	nQuantity:= 3, 
	nMBAddr:= 16#107, 
	cbLength:= 6, 
	pSrcAddr:= ADR(_aControlData[3,0]), 
	bExecute:= , 
	tTimeout:= T#1S, 
	bBusy=> , 
	bError=> , 
	nErrId=> );	
	

CASE _iSendReceiveState OF 
	0:
		_tonDelay2(IN:= FALSE);
		_iChannelIndex:= -1;
		FOR i := 0 TO 5 BY 1//进行读取指令的轮训
		DO
		 IF _aEnableSignal[i]//检测有控制指令发生
		 THEN
			 _iChannelIndex:=i;    
			END_IF 
		END_FOR
		IF _iChannelIndex>=4//有读取反馈指令
		THEN								
			IF NOT _aRead_VAR[_iChannelIndex].bBusy
			THEN
				_aRead_VAR[_iChannelIndex].bExecute := _aEnableSignal[_iChannelIndex];
				_iSendReceiveState := 10;	
			END_IF													
		END_IF			
		IF _iChannelIndex>=0 AND _iChannelIndex<=3//有控制触发指令
		THEN		
			IF  NOT _aWtirt_VAR[_iChannelIndex].bBusy 
			THEN
				_aWtirt_VAR[_iChannelIndex].bExecute := _aEnableSignal[_iChannelIndex];
				_iSendReceiveState := 10;
			END_IF
		END_IF
	10://等待读取响应			
		_tonDelay2(IN:= TRUE,PT:=T#3S);
		IF _tonDelay2.Q//超时
		THEN
			_iSendReceiveState:= 999;					
		END_IF				
		IF _iChannelIndex>=4
		THEN					
			IF _aRead_VAR[_iChannelIndex].bBusy
			THEN
				_iComNGCount := 0;
				_aEnableSignal[_iChannelIndex] := FALSE;
				_aRead_VAR[_iChannelIndex].bExecute := FALSE;
				_iSendReceiveState := 0;//等待下次触发
			ELSIF _aRead_VAR[_iChannelIndex].bError
			THEN
				_iComNGCount := _iComNGCount + 1;//错误次数加一
				IF _iComNGCount >= 3//重发多次失败
				THEN
					eOperErrorID := _aRead_VAR[_iChannelIndex].nErrId;
					_aRead_VAR[_iChannelIndex].bExecute := FALSE;
					_iSendReceiveState := 999;//进入错误发生状态
				ELSE
					_tonDelay1(in:=FALSE);
					_aRead_VAR[_iChannelIndex].bExecute:= FALSE;
					_iSendReceiveState := _iSendReceiveState + 1;
				END_IF						
			END_IF			
		END_IF				
		IF _iChannelIndex>=0 AND _iChannelIndex<=3		
		THEN	
			IF _aWtirt_VAR[_iChannelIndex].bBusy
			THEN
				_iComNGCount := 0;
				_aEnableSignal[_iChannelIndex] := FALSE;
				_aWtirt_VAR[_iChannelIndex].bExecute := FALSE;
				_iSendReceiveState := 0;//等待下次触发
			ELSIF _aWtirt_VAR[_iChannelIndex].bError
			THEN
				_iComNGCount := _iComNGCount + 1;//错误次数加一
				IF _iComNGCount >= 3//重发多次失败
				THEN
					eOperErrorID := _aWtirt_VAR[_iChannelIndex].nErrId;
					_aWtirt_VAR[_iChannelIndex].bExecute := FALSE;
					_iSendReceiveState := 999;//进入错误发生状态
				ELSE
					_tonDelay1(in:=FALSE);
					_aWtirt_VAR[_iChannelIndex].bExecute:= FALSE;
					_iSendReceiveState := _iSendReceiveState + 1;
				END_IF					
			END_IF				
		END_IF
	11://延时，进行补发操作
		_tonDelay1(in:=TRUE,pt:=T#300MS);				
		IF _tonDelay1.Q
		THEN
			_iSendReceiveState := 0;
		END_IF	
	999://错误状态，等待复位发生
		_xConnect_ERROR := TRUE;
		IF _fResetCheck.Q
		THEN	
			_aWtirt_VAR[0](bExecute := FALSE);
			_aWtirt_VAR[1](bExecute := FALSE);
			_aWtirt_VAR[2](bExecute := FALSE);
			_aWtirt_VAR[3](bExecute := FALSE);			
			_aRead_VAR[4](bExecute := FALSE);
			_aRead_VAR[5](bExecute := FALSE);
			_xConnect_ERROR := FALSE;
			_iComNGCount := 0;			
			_iSendReceiveState := 0;//重新开始
		END_IF
	ELSE
		;
END_CASE
END_ACTION

///{attribute 'tc_no_symbol'}
METHOD PROTECTED CyclicAction
VAR_OUTPUT
	xComplete: BOOL;
END_VAR
IF xAbort=0 THEN
    IF xFirstInvocation THEN
    (*
    * Staring
    * for then first (!) invocaion,
    * sample then input variables
    *)
			_xReadStatus := FALSE;
			_iCount := 0;
			_diCmdState := 0;
			_iAbortState := 0;
			_iNGCount := 0;
			_aRead_VAR[4].bExecute := FALSE;			
			_aRead_VAR[5].bExecute := FALSE;
			_aWtirt_VAR[0].bExecute:= FALSE;
			_aWtirt_VAR[1].bExecute:= FALSE;
			_aWtirt_VAR[2].bExecute:= FALSE;
			_aWtirt_VAR[3].bExecute:= FALSE;
			xFirstInvocation:=0;			
    END_IF    
    REPEAT 				
		  (**************************检查是否有硬件报错(检测总线是否报错)**********************************) 			
			IF stPara.strSlaveIP = '' 
			THEN
				eErrorID := RGI_14_ERROR.FLT_PARA;//参数配置错误
			END_IF
			//下面几个报警需要断驱动器的电才能消除报警
			IF st_IOData.I_DeviceERRORState <> 0 
			THEN
				eErrorID := RGI_14_ERROR.FLT_DEVICE_ERROR;//过热报警
			END_IF
		
			IF _xConnectError//检测子站是否有连接异常
			THEN
				eErrorID := RGI_14_ERROR.FLT_CONNECT;//子站通讯报警
			END_IF		
			//判断指令类型
			CASE eCmd OF
					//夹爪
					RGI_14_CMD.Cmd_Clamp,RGI_14_CMD.Cmd_Release://执行夹爪指令	
                        eClampActCmd := eCmd ;				
						CmdClampAction(xComplete=> xComplete);
					//绝对旋转	
					RGI_14_CMD.Cmd_RotateAbsClamp , RGI_14_CMD.Cmd_RotateAbsRelease ://执行旋转指令
						CmdRotateAction_ABS(xComplete=> xComplete);
					//相对旋转
					RGI_14_CMD.Cmd_RoratRelClamp , RGI_14_CMD.Cmd_RoratRelRelease://执行旋转指令
						CmdRotateAction_Ref(xComplete=> xComplete);
					//初始化
					RGI_14_CMD.Cmd_Org://执行回原点指令
						mCmdOrgAction(xComplete=> xComplete);
						
						
					ELSE
						;	
				END_CASE  
      UNTIL (TRUE)
	END_REPEAT
END_IF


IF xAbort OR xComplete OR eErrorID<>RGI_14_ERROR.NO_ERROR THEN    
    (*
    * Cleaning
    * => free as much allocated resources as possible
    *)    
    tOperationTimer(IN:=0);
END_IF
END_METHOD

///{attribute 'tc_no_symbol'}
METHOD PRIVATE FINAL HandleAbortedState
VAR_INPUT
END_VAR
VAR_OUTPUT
	xAgain: BOOL;
END_VAR
VAR
	xComplete: BOOL;
END_VAR
IF xAborted AND xResetRequest THEN
    eState:=STATE.RESETING;
    xAgain:=1;
ELSE
    xBusy:=0;
    xAborted:=1;
    //xResetRequest:=(xExecute=0);
    xAgain:=0;(* !!! *)
END_IF
END_METHOD

///{attribute 'tc_no_symbol'}
METHOD PRIVATE FINAL HandleAbortingState
VAR_OUTPUT
	xAgain: BOOL;
END_VAR
VAR
	xComplete: BOOL;
END_VAR
AbortAction(xComplete=> xComplete, eErrorID=> eErrorID);

IF eErrorID<>RGI_14_ERROR.NO_ERROR THEN
    eState:=STATE.INERROR;
    xAgain:=1;
ELSIF xComplete THEN
    eState:=STATE.ABORTED;
    xAgain:=1;
END_IF
END_METHOD

///{attribute 'tc_no_symbol'}
METHOD PRIVATE FINAL HandleDoneState
VAR_OUTPUT
	xAgain: BOOL;
END_VAR
//在运行过程中要是切换模式，再运行完成之后，检测到模式的切换，就需要回到初始位置，进行下一次执行准备
IF _xDone AND ((xExecute=0) OR ( _xModeChange AND NOT _xAutoOpe ) OR ( NOT xAutoMode AND NOT xDeviceRunning AND ( NOT _xAutoOpe OR _xHMIOpe))) THEN
	eState:=STATE.RESETING;
	xAgain:=1;
ELSE
	xBusy:=0;
	_xDone:=1;
	//xResetRequest:=(xExecute=0);
	xAgain:=0;(* !!! *)
END_IF
END_METHOD

///{attribute 'tc_no_symbol'}
METHOD PRIVATE FINAL HandleDormantState
VAR_OUTPUT
	xAgain: BOOL;
END_VAR

IF xExecute THEN
    xBusy:=1;
    eState:=STATE.EXECUTING;
    xAgain:=1;
END_IF

//下面两个报警一旦报警就需要发生
IF _xConnectError 
THEN//出现这个进行报警
	eERRORID := RGI_14_ERROR.FLT_CONNECT;//子站通讯报警
END_IF
IF st_IOData.I_DeviceERRORState <> 0//检测硬件是否报错
THEN
	eERRORID := RGI_14_ERROR.FLT_DEVICE_ERROR;//需要检查硬件，硬件有问题
END_IF

IF _fResetCheck.Q//清空报警
THEN
	eERRORID := RGI_14_ERROR.No_ERROR;
END_IF
(********************************等待手动操作******************************)
//初始化指令
_rHMIInit(CLK:= stOper.xHMInitButton AND eErrorID = RGI_14_ERROR.NO_ERROR AND NOT xAutoMode AND NOT xDeviceRunning AND NOT xIniting );
_rInit(CLK:= stOper.xInitControl AND eErrorID = RGI_14_ERROR.NO_ERROR AND ( xAutoMode OR  xDeviceRunning OR xIniting));
IF _rHMIInit.Q OR _rInit.Q
THEN
	eCmd := RGI_14_CMD.Cmd_Org;
	xExecute := TRUE;
END_IF

FOR ii := 1 TO 10 BY 1
DO 
	//夹紧轴夹紧控制
	_rHMIClamp[ii](CLK:= stOper.aHMIClampButton[ii] AND eErrorID = RGI_14_ERROR.NO_ERROR AND NOT xAutoMode AND NOT xDeviceRunning AND NOT xIniting);
	_rClamp[ii](CLK:= stOper.aClampControl[ii] AND eErrorID = RGI_14_ERROR.NO_ERROR AND ( xAutoMode OR xDeviceRunning OR xIniting ) );
	IF _rHMIClamp[ii].Q OR _rClamp[ii].Q
	THEN
		iTorqueSet :=stPosPara.aHMIClampiTorqueSet[ii];
		iSpeedSet := stPosPara.aHMIClampiSpeedSet[ii];
		iPosAngleSet := stPosPara.aHMIClampiPosAngleSet[ii];
		eCmd := RGI_14_CMD.Cmd_Clamp;
		xExecute := TRUE;
	END_IF	
	//夹紧轴松开指令
	_rHMIRelease[ii](CLK:= stOper.aHMIReleaseButton[ii] AND eErrorID = RGI_14_ERROR.NO_ERROR AND NOT xAutoMode AND NOT xDeviceRunning AND NOT xIniting);
	_rRelease[ii](CLK:= stOper.aReleaseControl[ii] AND eErrorID = RGI_14_ERROR.NO_ERROR AND ( xAutoMode OR  xDeviceRunning OR xIniting));
	IF _rHMIRelease[ii].Q OR _rRelease[ii].Q
	THEN
		iTorqueSet := stPosPara.aHMIReleasepiTorqueSet[ii];
		iSpeedSet :=stPosPara.aHMIReleasepiSpeedSet[ii];
		iPosAngleSet := stPosPara.aHMIReleasepiPosAngleSet[ii];
		eCmd := RGI_14_CMD.Cmd_Release;
		xExecute := TRUE;
	END_IF		
	//旋转轴关盖控制
	_rHMIRotateClamp[ii](CLK:= stOper.aHMIRotateClampButton[ii] AND eErrorID = RGI_14_ERROR.NO_ERROR AND NOT xAutoMode AND NOT xDeviceRunning AND NOT xIniting);
	_rRotateClamp[ii](CLK:= stOper.aRotateClampControl[ii] AND eErrorID = RGI_14_ERROR.NO_ERROR AND ( xAutoMode OR xDeviceRunning OR xIniting) );
	IF _rHMIRotateClamp[ii].Q OR _rRotateClamp[ii].Q
	THEN
		iTorqueSet := stPosPara.aHMIRotateiTorqueSet[ii];
		iSpeedSet := stPosPara.aHMIRotateClampiSpeedSet[ii];
		iPosAngleSet := stPosPara.aHMIRotateClampiPosAngleSet[ii];
		eCmd := RGI_14_CMD.Cmd_RotateAbsClamp;
		xExecute := TRUE;
	END_IF	
	//旋转轴松盖指令
	_rHMIRotateRelease[ii](CLK:= stOper.aHMIRotateReleaseButton[ii] AND eErrorID = RGI_14_ERROR.NO_ERROR AND NOT xAutoMode AND NOT xDeviceRunning AND NOT xIniting);
	_rRotateRelease[ii](CLK:= stOper.aRotateReleaseControl[ii] AND eErrorID = RGI_14_ERROR.NO_ERROR AND ( xAutoMode OR  xDeviceRunning OR xIniting ));
	IF _rHMIRotateRelease[ii].Q OR _rRotateRelease[ii].Q
	THEN
		iTorqueSet := stPosPara.aHMIRotateReleaseiTorqueSet[ii];
		iSpeedSet := stPosPara.aHMIRotateReleaseiSpeedSet[ii];
		iPosAngleSet := stPosPara.aHMIRotateReleaseiPosAngleSet[ii];
		eCmd := RGI_14_CMD.Cmd_RotateAbsRelease;
		xExecute := TRUE;
	END_IF	
	
	//相对旋转夹紧控制
	_rHMIRotateClampRef[ii](CLK:= stOper.aHMIRotateClampRefButton[ii] AND eErrorID = RGI_14_ERROR.NO_ERROR AND NOT xAutoMode AND NOT xDeviceRunning AND NOT xIniting);
	_rRotateClampRef[ii](CLK:= stOper.aRotateClampRefControl[ii] AND eErrorID = RGI_14_ERROR.NO_ERROR AND ( xAutoMode OR xDeviceRunning OR xIniting) );
	IF _rHMIRotateClampRef[ii].Q OR _rRotateClampRef[ii].Q
	THEN
		iTorqueSet := stPosPara.aHMIRotateRefiTorqueSet[ii];
		iSpeedSet := stPosPara.aHMIRotateClampRefiSpeedSet[ii];
		iPosAngleSet := stPosPara.aHMIRotateClampRefiPosAngleSet[ii];
		eCmd := RGI_14_CMD.Cmd_RoratRelClamp;
		xExecute := TRUE;
	END_IF
	//相对旋转松开控制
	_rHMIRotateReleaseRef[ii](CLK:= stOper.aHMIRotateReleaseRefButton[ii] AND eErrorID = RGI_14_ERROR.NO_ERROR AND NOT xAutoMode AND NOT xDeviceRunning AND NOT xIniting);
	_rRotateReleaseRef[ii](CLK:= stOper.aRotateReleaseRefControl[ii] AND eErrorID = RGI_14_ERROR.NO_ERROR AND ( xAutoMode OR xDeviceRunning OR xIniting ) );
	IF _rHMIRotateReleaseRef[ii].Q OR _rRotateReleaseRef[ii].Q
	THEN
		iTorqueSet := stPosPara.aHMIRotateReleaseRefiTorqueSet[ii];
		iSpeedSet := stPosPara.aHMIRotateReleaseRefiSpeedSet[ii];
		iPosAngleSet := stPosPara.aHMIRotateReleaseRefiPosAngleSet[ii];
		eCmd := RGI_14_CMD.Cmd_RoratRelRelease;
		xExecute := TRUE;
	END_IF
	
END_FOR
END_METHOD

METHOD PRIVATE FINAL HandleErrorState
VAR_OUTPUT
	xAgain: BOOL;
END_VAR
IF xError THEN
	IF eErrorID < RGI_14_ERROR.FLT_ClAMP_CLAMPFAIL//正常执行报警
	THEN
		IF xResetRequest OR NOT xExecute//按照正常逻辑进行处理复位处理就可以
		THEN
				eState:=STATE.RESETING;
				xAgain:=1;
		END_IF
	ELSE//操作失败报警（有可能需要进行程序跳步处理，此时，在自动模式下不允许被复位掉，防止，程序异常死机）
		IF ( NOT xAutoMode AND xIniting ) OR xAutoMode
		THEN 
			IF NOT xExecute//按照正常逻辑进行处理复位处理就可以
			THEN 
				eState:=STATE.RESETING;
				xAgain:=1;
			END_IF
		ELSE
			IF xResetRequest OR NOT xExecute//按照正常逻辑进行处理复位处理就可以
			THEN
				eState:=STATE.RESETING;
				xAgain:=1;
			END_IF
		END_IF
	END_IF
ELSE
	xBusy:=0;
	xError:=1;    
	xAgain:=0;(* !!! *)
END_IF
END_METHOD

///{attribute 'tc_no_symbol'}
METHOD PRIVATE FINAL HandleExecutingState
VAR_OUTPUT
	xAgain: BOOL;
END_VAR
VAR
	xComplete: BOOL;
END_VAR
IF xAbort=0 THEN   
    CyclicAction(xComplete=> xComplete);
END_IF

IF eErrorID<>RGI_14_ERROR.NO_ERROR THEN
    eState:=STATE.INERROR;
    xAgain:=1;
ELSIF xAbort THEN
    eState:=STATE.ABORTING;
    xAgain:=1;
ELSIF xComplete THEN
    eState:=STATE.DONE;
    xAgain:=1;
END_IF
END_METHOD

///{attribute 'tc_no_symbol'}
METHOD PRIVATE FINAL HandleResettingState
VAR_OUTPUT
	xAgain: BOOL;
END_VAR
VAR
	xComplete: BOOL;
END_VAR
ResetAction(xComplete=> xComplete);

IF xComplete THEN
	xExecute:=0;//清除输入指令 
    xBusy:=0;
    _xDone:=0;
    xError:=0;
    xAborted:=0;
    eErrorID:=RGI_14_ERROR.NO_ERROR;
    eState:=STATE.DORMANT;
    xFirstInvocation:=1;
    xAgain:=0;(* !!! *)
END_IF
END_METHOD

METHOD PROTECTED mCmdOrgAction
VAR_OUTPUT
	xComplete: BOOL;
END_VAR
VAR
	thebn: INT;
END_VAR
// return the real actual fault number
IF eErrorID <> RGI_14_ERROR.NO_ERROR
THEN
  RETURN;  
END_IF

CASE _diCmdState OF
	0://a相关数据初始化
		xRefOk := FALSE;//因为需要重新初始化，所以需要清除回原点完成标志位	
		_tonDelay(IN:= FALSE);
		st_IOData.O_RotateAngleLSet := 0;
		st_IOData.O_RotateAngleHSet := 0;
		st_IOData.O_RotateRelAngle := 0;
		IF NOT _aRead_VAR[5].bExecute THEN//没有读取任务
			_diCmdState := _diCmdState + 1;
		END_IF			
		
	1://初始化赋值
		_tonDelay(IN:= TRUE,pt:=T#20MS);
		st_IOData.O_Init := 16#A5;//触发回原点指令
		IF _tonDelay.Q//错开刷新时序
		THEN  
			_tonCmdTimeout(in:=FALSE); 
			_tonDelay(IN:=FALSE);
			_aEnableSignal[0]:=TRUE;   
			_diCmdState := _diCmdState+1;
		END_IF
		
	2://等待使能失效被响应	
		_tonCmdTimeout(IN:= _aEnableSignal[0],pt:=T#2S);
		_tonDelay(IN:=NOT _aEnableSignal[0],PT:=T#200MS);
		IF _tonDelay.Q
		THEN
			_tonCmdTimeout(in:=FALSE);
			SysMemSet(ADR(_aFeedbackData),0,SIZEOF(_aFeedbackData));
			_diCmdState := _diCmdState +1; 
		END_IF	
		
		IF _iSendReceiveState = 999//指令超时报错
		THEN
			eErrorID := RGI_14_ERROR.FLT_ORGCMD_TIMEOUT;		
			_diCmdState := 999;
		END_IF  
		
	3://设置读取数据反馈	 
		_tonCmdTimeout(in:=FALSE);
		_tonTimeout(in:=TRUE,pt:=T#10S); 
		_tonDelay(IN:= FALSE);
		_aEnableSignal[5] := TRUE;//读取状态信息
		_diCmdState := _diCmdState +1; 
		
	4://等待数据接收完成		
		_tonTimeout(in:=TRUE,pt:=T#10S); 
		_tonCmdTimeout(IN:= TRUE,pt:=T#2S); 
		IF NOT _aEnableSignal[5]//等待电动夹爪响应 
		THEN			
			_tonDelay(IN:= TRUE,pt:=T#40MS);//设置刷新周期
			IF st_IOData.I_ClampInit = 1 (*AND st_IOData.I_RotateInit = 1 *)  //判断是否初始化成功
			THEN
				_tonCmdTimeout(in:=FALSE);
				_tonDelay(IN:= FALSE);
				_tonTimeout(in:=FALSE);  
				_diCmdState := 100;
				xRefOk := TRUE;//标记回原点成功
				xComplete := 1;
			END_IF
			IF _tonDelay.Q
			THEN
				_diCmdState := 3;
			END_IF
		END_IF	
		IF _iSendReceiveState = 999//回原点指令响应超时
		THEN
			eErrorID := RGI_14_ERROR.FLT_ORGCMD_TIMEOUT;		
			_diCmdState := 999;
		END_IF	
		IF _tonTimeout.Q//回原点动作超时
		THEN
			eErrorID := RGI_14_ERROR.FLT_ORG_TIMEOUT;
			_diCmdState := 999;
		END_IF			
	ELSE
		;
END_CASE
END_METHOD

///{attribute 'tc_no_symbol'}
METHOD PROTECTED ResetAction
VAR_OUTPUT
	xComplete: BOOL;
END_VAR
(*
* Cleaning
* => free all allocated resources
* => reinitialize instance variables
*)
tOperationTimer(IN:=0);

// init command state
_diCmdState := 0;
_iAbortState := 0;
_tonCmdTimeout(in:=FALSE);
_tonTimeout(in:=FALSE);
_tonDelay(IN:=FALSE);
_xRotateFinish := FALSE;
_xModeChange := FALSE;
_xReadStatus :=  TRUE;
_iNGCount := 0;

//清除触发标志位
FOR i:= 0 TO 5 BY 1
DO
	_aEnableSignal[i] := FALSE;
END_FOR
FOR i:= 4 TO 5 BY 1
DO
	_aRead_VAR[i].bExecute:= FALSE; 
END_FOR
FOR i:= 0 TO 3 BY 1
DO
	_aWtirt_VAR[i].bExecute:= FALSE; 
END_FOR

FOR ii :=1 TO 10 DO
	//手头指令清除
	stOper.aHMIClampButton[ii]:=FALSE;
	stOper.aHMIReleaseButton[ii]:=FALSE;
	stOper.aHMIRotateClampButton[ii]:=FALSE;
	stOper.aHMIRotateClampRefButton[ii]:=FALSE;
	stOper.aHMIRotateReleaseButton[ii]:=FALSE;
	stOper.aHMIRotateReleaseRefButton[ii]:=FALSE;
	stOper.xHMInitButton:=FALSE;	
	//自动指令操作
	stOper.aClampControl[ii]:=FALSE;
	stOper.aReleaseControl[ii]:=FALSE;
	stOper.aRotateClampControl[ii]:=FALSE;
	stOper.aRotateClampRefControl[ii]:=FALSE;
	stOper.aRotateReleaseControl[ii]:=FALSE;
	stOper.aRotateReleaseRefControl[ii]:=FALSE;
	stOper.xInitControl:=FALSE;	
END_FOR



//清除触发标志位
xComplete:=1;
END_METHOD

END_FUNCTION_BLOCK

// ---- POUs/003_FB/03_TURINRobotFB/FB_TURINContorl.TcPOU
FUNCTION_BLOCK FB_TURINContorl
VAR_INPUT
	xManuMode : BOOL;//设备手动模式显示
	xAutoRunning : BOOL;//设备是否自动运行
	xEStop : BOOL;//设备急停信号
	xMovePermit : BOOL;//运行允许
	xReset      : BOOL;//复位按钮
	xStart      : BOOL;//启动按钮
	xStop      : BOOL;//停止按钮
	xPause      : BOOL;//暂停按钮
	xContinue      : BOOL;//继续按钮
	xInitExte   : BOOL;//初始化执行指令	
	xClearInitedFlag : BOOL;
	stPara       : ST_Sys_Para;//系统参数	
	pSysToRobot : ARRAY [0..3] OF WORD;//plc to robot 数据
	pSysFromRobot : ARRAY [0..3] OF WORD;//plc from robot 数据
END_VAR
VAR_OUTPUT
	xInitedFlag : BOOL;//初始化完成
	xInitFinish : BOOL;
	iCurrentStatus : INT; 
	eErrID  : TURIN_ERROR;
END_VAR
VAR_IN_OUT	
	stData : ST_TURINROBOT_Data;//机器人信号数据
END_VAR
VAR
	{attribute 'tc_no_symbol'}
	_iInitState , _iStartState , _iStopStateb , _iConnectState ,_iEpsonState: INT;//初始化状态
	{attribute 'tc_no_symbol'}
	_ton1 , _ton2 , _ton3 , _ton4 , _connectTon : TON;//
	{attribute 'tc_no_symbol'}
	_xInitFinish : BOOL;
	{attribute 'tc_no_symbol'}
	_fResetCheck : F_TRIG;
	{attribute 'tc_no_symbol'}
	_xConnectError : BOOL;//有连接报错发生
	{attribute 'tc_no_symbol'}
	_rManualMode : R_TRIG;
	{attribute 'tc_no_symbol'}
	_fManualMode : f_TRIG;
	{attribute 'tc_no_symbol'}
	_tonInit : TON;
	{attribute 'tc_no_symbol'}
	_tonPWM1 , _tonPWM2 : TON;
	{attribute 'tc_no_symbol'}
	_rTrig_Paused			:R_TRIG;
	{attribute 'tc_no_symbol'}
	_rTrig_Continue		:R_TRIG;
	{attribute 'tc_no_symbol'}
	_rTrig_Init				:R_TRIG;
	{attribute 'tc_no_symbol'}
	_tonCmd : TON ;
	{attribute 'tc_no_symbol'}
	_tonDelay : TON ;
	{attribute 'tc_no_symbol'}
	_iNGCount : INT ;
	{attribute 'tc_no_symbol'}
	_irxState: INT := 0;
	{attribute 'tc_no_symbol'}
	_aRead_VAR :ARRAY [1..2] OF FB_MBReadInputs;
	{attribute 'tc_no_symbol'}
	_aWirte_VAR: FB_MBWriteCoils;
END_VAR


DataMap();//系统IO映射
SYSError();

//Start();//初始化流程已经启动机械手
Stop();
Init();
Connect();
CommonHandle();

ACTION CommonHandle:
//对应HMI显示窗：5-报警中；4-停止中；3-未初始化；2-运行中；
IF (eErrID <> TURIN_ERROR.NO_ERROR) AND  (eErrID <> TURIN_ERROR.FLT_NO_INIT)
THEN
	iCurrentStatus := 5;
ELSIF ( NOT stData.i_Running AND xInitFinish )
THEN
	iCurrentStatus := 4;
ELSIF NOT xInitFinish
THEN
	iCurrentStatus := 3;
ELSIF stData.i_Running
THEN
	iCurrentStatus := 2;
ELSE
	iCurrentStatus := 4;	
END_IF
END_ACTION

ACTION Connect:
//读取机械手数据
_aRead_VAR[1](
	sIPAddr:= stPara.strSlaveIP, 
	nTCPPort:= stPara.iSlavePort, 
	nUnitID:= stPara.bySlaveID, 
	nQuantity:= 32, 
	nMBAddr:= 0, 
	cbLength:= 32, 
	pDestAddr:= ADR(pSysFromRobot[0]), 
	bExecute:= stSysPulse.xP10ms, //fbMachine[1].xStart, //
	tTimeout:=T#1S , 
	bBusy=> , 
	bError=> , 
	nErrId=> , 
	cbRead=> );

_aRead_VAR[2](
	sIPAddr:= stPara.strSlaveIP, 
	nTCPPort:= stPara.iSlavePort, 
	nUnitID:= stPara.bySlaveID, 
	nQuantity:= 32, 
	nMBAddr:= 36, 
	cbLength:= 32, 
	pDestAddr:= ADR(pSysFromRobot[2]), 
	bExecute:= stSysPulse.xP10ms, //fbMachine[1].xStart, //
	tTimeout:=T#1S , 
	bBusy=> , 
	bError=> , 
	nErrId=> , 
	cbRead=> );
	
//写入机械手数据
_aWirte_VAR(
	sIPAddr:=stPara.strSlaveIP , 
	nTCPPort:=stPara.iSlavePort , 
	nUnitID:=stPara.bySlaveID , 
	nQuantity:= 64, 
	nMBAddr:= 24, 
	cbLength:= 64, 
	pSrcAddr:= ADR(pSysToRobot[0]), 
	bExecute:=stSysPulse.xP10ms ,  
	tTimeout:=T#1S , 
	bBusy=> , 
	bError=> , 
	nErrId=> );
END_ACTION

ACTION DataMap:
	(********************************************from robot 数据映射*********************************************)
	stData.i_EStopOn       := pSysFromRobot[0].0;	
  stData.i_Ready         := pSysFromRobot[2].0;  
	stData.i_Running       := pSysFromRobot[1].8;
	stData.i_Paused        := pSysFromRobot[1].1;
	stData.i_Error         := pSysFromRobot[2].3;
	stData.i_SError        := pSysFromRobot[2].4;
	stData.i_Waning        := pSysFromRobot[2].5;
	stData.i_MotorsOn      := pSysFromRobot[2].6;
	stData.i_AutoMode      := pSysFromRobot[0].2;
	stData.i_TeachMode     := NOT pSysFromRobot[0].2;
	stData.i_CmdError      := pSysFromRobot[2].9;

	(********************************************to robot 数据映射*********************************************)
	pSysToRobot[0].0 := stData.o_Start;    
	pSysToRobot[0].1 := stData.o_Stop OR stData.o_Pause;        
	pSysToRobot[0].2 := stData.o_Pause;       
	pSysToRobot[0].3 := stData.o_Continue;    
	pSysToRobot[0].4 := stData.o_Reset;      
	pSysToRobot[0].5 := stData.o_Init; 
	pSysToRobot[0].6 := stData.o_SetMotorsOff;
	pSysToRobot[0].7 := stData.o_RunCondition:=NOT xMovePermit;
END_ACTION

ACTION Init:
_rTrig_Init(CLK:= xInitExte, Q=> );
(*IF 	(NOT (eErrID =E_Epson_ERROR.FLT_NO_INIT)
	AND
		NOT (eErrID =E_Epson_ERROR.NO_ERROR))
	OR
		_tonInit.Q//初始化超时
THEN
		_iInitState := 0;	
END_IF
IF xManuMode//手动模式处于
THEN	
	CASE _iInitState OF 
		0://执行条件是不能有错误发生，有错误发生，优先去处理错误
			IF _rTrig_Init.Q AND (eErrID =E_Epson_ERROR.NO_ERROR OR eErrID =E_Epson_ERROR.FLT_NO_INIT)
			THEN
				_xInitFinish := FALSE;
				xInitFinish:=FALSE;
				_iInitState := 1;
			END_IF
		1://ROBOT Paused
			IF  stData.i_Paused THEN
				stData.o_Continue := TRUE;
			END_IF
			IF NOT stData.i_Paused THEN
				IF stData.i_Running THEN
					_iInitState :=3;	
				END_IF
				IF NOT stData.i_Running THEN
					_iInitState :=2;	
				END_IF	
				stData.o_Continue := FALSE;		
			END_IF
		2://ROBOT NOT Running	
					_iInitState :=4;				
		3://ROBOT Running	
				stData.o_Stop := TRUE;	
				IF NOT stData.i_Running THEN
					_iInitState :=4;	
				END_IF		
		4://进行信号准备
			//xInitExte := FALSE;
			stData.o_Stop := FALSE;
			stData.o_Pause := FALSE;		
      stData.o_Continue := FALSE;	
			_iInitState := 5;	
		5://等待robot Motor on
			stData.o_SetMotorsOn := TRUE;
			stData.o_SetMotorsOff := FALSE;			
			IF stData.i_MotorsOn
			THEN		
				stData.o_SetMotorsOn := FALSE;
				stData.o_SetMotorsOff := FALSE;		
				_iInitState := 6;
			END_IF		
		6://程序启动成功
			stData.o_Start := TRUE;
			IF stData.i_Running//代表程序已经启动起来
			THEN	
				//检测启动程序是否正确
				IF stData.o_SelProg1 = stData.i_CurrProg1 AND 	
					 stData.o_SelProg2 = stData.i_CurrProg2 AND 
					 stData.o_SelProg4 = stData.i_CurrProg4
				THEN	
					xInitedFlag := TRUE;	
					_iInitState := 100;
				ELSE
					stData.o_Start := FALSE;
					_iInitState := 0;
				END_IF					
			END_IF			
	
		100://等待外部响应完成，回到起始状态
				stData.o_Start := FALSE;
			IF stData.i_AtHome
			THEN	
				_xInitFinish := TRUE;
				_iInitState := 110;
			END_IF
		110:
			IF _xInitFinish THEN
				xInitFinish:=TRUE;
				_iInitState := 0;
			END_IF
		ELSE
			;
	END_CASE
END_IF
*)
IF xManuMode//手动模式处于
THEN	
	CASE _iInitState OF 
		0://触发信号
		IF _rTrig_Init.Q THEN
				xInitFinish:=FALSE;
				xInitExte := FALSE;
				_iNGCount := 0 ;
				_iInitState := _iInitState + 1;
		END_IF
    1://判断条件是否满足
		IF not stData.i_EStopOn THEN 
				_iInitState := 999;
				eErrID := TURIN_ERROR.FLT_ESTOPON ;
		ELSIF eErrID <> TURIN_ERROR.NO_ERROR THEN
				_iInitState := 999;
		ELSIF NOT stData.i_AutoMode THEN 
				_iInitState := 999;	
				eErrID := TURIN_ERROR.FLT_AUTOMODE ;		
		ELSE 

				_iInitState := _iInitState + 1;
		END_IF

		2://检测是否运行中
		 IF stData.i_Running THEN 
		    stData.o_Stop := TRUE ;		
		 ELSE
				_iInitState:=_iInitState + 1;
				stData.o_Stop := FALSE ;	
		 END_IF		
		
		3://跳转首行
				_tonDelay(IN:=TRUE,PT:=T#3S);
				stData.o_Init:=TRUE;
		 IF stData.i_Ready THEN 
			 	stData.o_Init:=FALSE;
			 	_iInitState := _iInitState + 1;
		 ELSIF _tonDelay.Q THEN
				_tonDelay(IN:=FALSE);
				stData.o_Init:=False;
				stToRobotZero.iMoveMode:=stToRobotZero.iMoveMode+1;
				eErrID := TURIN_ERROR.FLT_SYSREADY ;				
				_iInitState := 999;
		 END_IF

		4://__________
				_tonDelay(IN:=TRUE,PT:=T#200MS);
				IF _tonDelay.Q  THEN 
				_tonDelay(IN:=FALSE);
				_iInitState := _iInitState + 1;
				END_IF
	  5://触发停止信号
				_tonDelay(IN:=TRUE,PT:=T#200MS);
		    stData.o_Stop := TRUE ;
		 IF _tonDelay.Q  THEN 
				_tonDelay(IN:=FALSE);
		    stData.o_Stop := FALSE ;

				_iInitState := _iInitState + 1;
		 END_IF
		 6://检测不在运行中
				_tonDelay(IN:=TRUE,PT:=T#200MS);
		 IF _tonDelay.Q THEN 
				 IF  NOT stData.i_Running THEN 
						_tonDelay(IN:=FALSE);
						_iInitState := _iInitState + 1;
				 ELSE 
						  _tonDelay(IN:=FALSE);
							eErrID := TURIN_ERROR.FLT_SYSREADY ;
							_iInitState := 999;			 
				 END_IF
		 END_IF
	 
		 7://触发启动信号
				_tonDelay(IN:=TRUE,PT:=T#500MS);
		    stData.o_Start := TRUE ;
		 IF _tonDelay.Q THEN 
				_tonDelay(IN:=FALSE);
		    stData.o_Start := FALSE ;
				_iInitState := _iInitState + 1;
		 END_IF		 
		 8://判断是否为Running
		  IF stData.i_Running  THEN 
				_iInitState := _iInitState + 1;
			ELSE 
				_iInitState := 4 ;
				_iNGCount := _iNGCount +1 ;
				IF _iNGCount>3 THEN 
					_iNGCount := 0 ;
					eErrID := TURIN_ERROR.FLT_No_Runing ;
				  _iInitState := 999;
				END_IF
			END_IF
		  9://初始化完成
				xInitFinish:=TRUE;
				  _iInitState := 999;
      999://
				  _iInitState := 0;
		 
		 
		 
		 
		 
		 
		 
	END_CASE
END_IF
END_ACTION

ACTION Start:
//启动主流程
CASE _iStartState OF 
	0://等待设备处于自动运行状态
		IF xAutoRunning AND eErrID = TURIN_ERROR.NO_ERROR
		THEN
			_iStartState := _iStartState + 1;
		END_IF
	1://检测是否满足启动条件
		IF NOT _xInitFinish
		THEN
			eErrID := TURIN_ERROR.FLT_NO_INIT;	
			_iStartState := 0;		
		END_IF	
		IF eErrID = TURIN_ERROR.NO_ERROR
		THEN
			_iStartState := _iStartState + 1;
		END_IF
	2://等待开始启动
		IF NOT stData.o_Stop
		THEN
			_iStartState := _iStartState + 1;
		END_IF	
	3://robot modeon
		stData.o_SetMotorsOn := _tonPWM1.Q;
		stData.o_SetMotorsOff := FALSE;
		_ton1(IN:=stData.i_MotorsOn,PT:=T#200MS);
		IF _ton1.Q
		THEN			
			_ton1(IN:=FALSE);
			_iStartState := 10;
		END_IF	
	10://程序启动成功
		stData.o_Start := _tonPWM1.Q; 
		IF stData.i_Running
		THEN				
			stData.o_Start := FALSE;
			_iStartState := 100;//代表启动完成	
		END_IF
	ELSE
		;		
END_CASE
END_ACTION

ACTION Stop:
//robot停止信号控制

	_rTrig_Paused(CLK:=NOT xAutoRunning , Q=> );
	_rTrig_Continue(CLK:=xAutoRunning , Q=> );
	
(*IF _xInitFinish//已经初始化完成
THEN
	stData.o_Pause := ( _rTrig_Paused.Q OR  NOT xMovePermit ) AND NOT stData.i_Paused ;	
	stData.o_Continue := (_rTrig_Continue.Q AND xMovePermit ) AND stData.i_Paused ;   
END_IF
*)
//关联操作按钮
stData.o_Reset := xReset;
IF  xPause OR xStop OR _rTrig_Paused.Q THEN 
	 stData.o_Pause := TRUE ;
ELSE 
	 stData.o_Pause := FALSE ;
END_IF
IF stData.i_Paused THEN 
	 stData.o_Continue := xStart;
ELSE 
	 stData.o_Start := xStart ;
END_IF
END_ACTION

ACTION SYSError:

_ton3(in:= NOT _ton4.Q,PT:= T#300MS);
_ton4(in:= _ton3.Q,PT:= T#300MS);
stData.o_Reset := xReset AND _ton3.Q;//产生脉冲信号
IF eErrID <> TURIN_ERROR.NO_ERROR
THEN
	stData.o_Reset := xReset AND _ton3.Q;//产生脉冲信号
END_IF

//Epson cmd Status	

IF NOT stData.i_EStopOn 
THEN
			eErrID := TURIN_ERROR.FLT_ESTOPON;//检测是否有急停产生
ELSE
CASE _iEpsonState OF 
		
	0://检测是否有指令错误发生
		IF stData.i_CmdError  THEN
			eErrID := TURIN_ERROR.FLT_CMDERROR;
			_iEpsonState:=0;					
		END_IF
		IF (eErrID <> TURIN_ERROR.FLT_CMDERROR) THEN
			_iEpsonState:=1;
		END_IF
	1://检测是否有错误发生
		IF stData.i_Error  THEN
			eErrID := TURIN_ERROR.FLT_ERROR;
			_iEpsonState:=0;					
		END_IF
		IF (eErrID <> TURIN_ERROR.FLT_ERROR) THEN
			_iEpsonState:=2;
		END_IF
	2://检测是否有系统错误产生
		IF stData.i_SError  THEN
			eErrID := TURIN_ERROR.FLT_SERROR;
			_iEpsonState:=0;					
		END_IF
		IF (eErrID <> TURIN_ERROR.FLT_SERROR) THEN
			_iEpsonState:=3;
		END_IF
	3://检测是否有警告发生
		IF stData.i_Waning THEN
			eErrID := TURIN_ERROR.FLT_SERROR;
			_iEpsonState:=0;					
		END_IF	
		IF (eErrID <> TURIN_ERROR.FLT_SERROR) THEN
			_iEpsonState:=4;
		END_IF
	4://检测配置参数是否不正确
		IF stPara.iSlavePort = 0 OR 
			 stPara.bySlaveID = 0  OR
			 stPara.strSlaveIP = ''
		THEN
				eErrID := TURIN_ERROR.FLT_PARA;
				_iEpsonState:=0;		
		END_IF	
		IF (eErrID <> TURIN_ERROR.FLT_PARA) THEN
			_iEpsonState:=5;
		END_IF	

	5://检测是否有连接错误
		IF _xConnectError 
		THEN
			eErrID := TURIN_ERROR.FLT_CONNECTERROR;
			_iEpsonState:=0;		
		END_IF
		IF (eErrID <> TURIN_ERROR.FLT_CONNECTERROR) THEN
			_iEpsonState:=7;
		END_IF		
	
	6://检测是否Ready
		IF xAutoRunning AND xInitFinish AND NOT stData.i_Running THEN
			eErrID := TURIN_ERROR.FLT_No_Runing;
			_iEpsonState:=0;					
		END_IF	
		IF (eErrID <> TURIN_ERROR.FLT_No_Runing) THEN
			_iEpsonState:=7;
		END_IF

	7://检测是否自动
		IF NOT xManuMode AND NOT stData.i_AutoMode THEN
			eErrID := TURIN_ERROR.FLT_AUTOMODE;
			xInitFinish:=FALSE;
			_iEpsonState:=0;					
		END_IF	
		IF (eErrID <> TURIN_ERROR.FLT_AUTOMODE) THEN
			_iEpsonState:=8;
		END_IF
	
	8://检测是否初始化完成
		IF NOT xManuMode AND NOT xInitFinish AND NOT xInitExte THEN
			eErrID := TURIN_ERROR.FLT_NO_INIT;
			_iEpsonState:=0;					
		END_IF	
		IF (eErrID <> TURIN_ERROR.FLT_NO_INIT) THEN
			_iEpsonState:=9;
		END_IF	
	
	9://检测是否初始化超时
		IF _tonInit.Q THEN
			eErrID := TURIN_ERROR.FLT_NO_INIT;
			_iInitState := 0;	//初始化流程归零	
			_iEpsonState:=0;					
		END_IF	
		IF (eErrID = TURIN_ERROR.NO_ERROR ) THEN
			_iEpsonState:=100;
		END_IF
	
100:	//检测无错误
		eErrID := TURIN_ERROR.NO_ERROR;
		_iEpsonState:=0;		
	
	END_CASE
	END_IF

//复位初始化完成
		IF NOT stData.i_AutoMode THEN
			xInitFinish:=FALSE;			
		END_IF	
	
//清除错误
IF xReset
THEN 
	_xConnectError := FALSE;//复位连接错误
	_iEpsonState:=0;
	eErrID := TURIN_ERROR.NO_ERROR;
END_IF

//初始化超时
_tonInit(IN:=_iInitState <> 0 ,PT:=T#20S);
END_ACTION

END_FUNCTION_BLOCK

// ---- POUs/001_Station/S10_BeltCarrying.TcPOU
PROGRAM S10_BeltCarrying
VAR
	//工站
	station					: REFERENCE TO FB_Station:=fbstation[10];
	//气缸
	
	//伺服
	fbROTAxisMove	 :REFERENCE TO FB_Axis:=fbAxis[16];	//	出料线体伺服
	
	//延时
	arTonDelay :ARRAY[1..20] OF TON;
	//返回值
	UdiReturnValue :ARRAY[1..20] OF UDINT;
	//过程记录
	tsModuleProcess:ARRAY[1..gc_ModuleProNo] OF DUT_Process;
	xClearModuleProcessDone:BOOL;
	bClearProcessStep	:BYTE;
	i,t: INT;
	bCounter:BYTE;
	 //报警屏蔽
	_AlarmDisable: BOOL;
	//首次循环
	_FirstCycle: ARRAY[1..10]OF BOOL;
	// //入料允许
	xBeltMovingEnable: BOOL;
	wActionCalibration: WORD;
	// 起始位置
	rStartPoition: ARRAY[0..8] OF REAL;
	// 结束位置
	rEndPoition:ARRAY[0..8] OF  REAL;
	NextPosR_TRIG: R_TRIG;
	tes: REAL;
	// 深孔板检测传感器
	xBoxSensorReached: ARRAY[1..2] of BOOL;
	xNotStop: BOOL;
	// 间距
	rcalcPos: ARRAY[0..7] OF REAL;
	//平均数
	raverage:REAL;
	_xFirstCycle: BOOL;
END_VAR

A_Input();
Alarm();
Delay();
FlowAuto();
FlowInit();
General();
ILC();
TipAuto();
TipManual();
Z_Output();

ACTION A_Input:
//气缸
//传感器
xBoxSensorReached[1]:=IxBeltEntryBoxCheckSensor2	;//	皮带线入口处¶深孔板检测传感器1
xBoxSensorReached[2]:=IxBeltEntryBoxCheckSensor1	;//	皮带线入口处¶深孔板检测传感器2

//允许进料
xBeltMovingEnable:=sModbus_200SMART.iBeltEnterEnable =1;
END_ACTION

ACTION Alarm:
//
station.adwAlarm[1].00:=station.xInitTimeout;	  			//S09CardCarrying 初始化超时
END_ACTION

ACTION Delay:
arTonDelay[01](IN:= , PT:=T#0.1S , Q=> , ET=> );
(*arTonDelay[02](IN:=  , PT:=T#1S , Q=> , ET=> );*)//已被使用
(*arTonDelay[03](IN:=   , PT:=T#1S , Q=> , ET=> );*)//已被使用
arTonDelay[04](IN:= , PT:=T#0.1S , Q=> , ET=> );
arTonDelay[05](IN:= , PT:=T#0.1S , Q=> , ET=> );
arTonDelay[06](IN:= , PT:=T#0.1S , Q=> , ET=> );
arTonDelay[07](IN:= , PT:=T#0.1S , Q=> , ET=> );
arTonDelay[08](IN:= , PT:=T#0.1S , Q=> , ET=> );
arTonDelay[09](IN:= , PT:=T#0.1S , Q=> , ET=> );
arTonDelay[10](IN:= NOT fbROTAxisMove.xbusy , PT:=T#0.1S , Q=> , ET=> );//TipAuto使用
END_ACTION

ACTION FlowAuto:

//-----------------------------------------初始化是否完成判断----------------------------------------------
IF NOT station.xInitDone 
THEN
 	station.iStepAuto:=0;
 	station.xDone:=FALSE;
ELSIF station.xRunning   OR 
(tsModuleProcess[1].xProcessStarted AND NOT tsModuleProcess[1].xProcessCompleted) OR//皮带线伺服移动
(tsModuleProcess[2].xProcessStarted AND NOT tsModuleProcess[2].xProcessCompleted)  //皮带线回原点
THEN
//-----------------------------------------动作步骤--------------------------------------------------------
CASE station.iStepAuto OF	  
	0: //----Home Step，等待启动----
		IF station.xDisabled 
			AND station.xCanRun 
			AND NOT fbMachine[1].xStopped 
			AND NOT station.xSingleRunning 
		THEN
			station.xDone:=TRUE;
		END_IF
		
		IF  station.xSingleRunning 
			OR station.xCanRun 
			//AND NOT station.xDone 
			AND NOT station.xDisabled 
			AND NOT fbMachine[1].xStopped
		THEN
			station.xCycleEnable:=TRUE;
			//station.xDone:= FALSE;  
			
			station.iStepAuto:= 10;
		END_IF
    10: //复位数据 
			IF  station.xSingleRunning THEN
				 FOR i:=1 TO gc_ModuleProNo BY 1 DO
						 MEMSET(ADR(tsModuleProcess[i]),0,SIZEOF(tsModuleProcess[i]));
				 END_FOR
			END_IF
			station.iStepAuto:=15;
	15://等待工位完成信号
		IF  NOT  fbMachine[1].xTryRun AND   NOT station.xSingleRunning THEN 
			IF  S07_BoxCarrying.station.xDone  AND 
				S09_CardCarrying.station.xDone  AND (xBeltMovingEnable OR S11_Packing.station.xDisabled ) THEN
					station.iStepAuto:=25;
			END_IF
		ELSE
		 			station.iStepAuto:=25;
		END_IF
	25://不允许各工位放料
				station.xDone :=FALSE;
				station.iStepAuto:=80;	   
	80://
				tsModuleProcess[1].xProcessNotStarted:=TRUE;
			  rStartPoition[t]:=fbROTAxisMove.rActPos;
				station.iStepAuto:=90;
	90://储存当前位置
			stData.Axis[16].rMovePosition[3]:=fbROTAxisMove.rActPos;
			station.iStepAuto:=95;
	95://读取原点偏移量
		 IF NOT _xFirstCycle THEN
		   stData.Axis[16].rMovePosition[2] := stData.Axis[16].rMovePosition[1] ;
		   _xFirstCycle := TRUE ;
		 END_IF
		   station.iStepAuto:=110;	
	110://数据更新 位置
				 tsModuleProcess[1].xProcessStarted:=TRUE;
				 stData.Axis[16].rMovePosition[2] := stData.Axis[16].rMovePosition[2] +stData.Axis[16].rRelativeDistance ;
				 arTonDelay[03](IN:= FALSE , PT:=T#50MS , Q=> , ET=> );
				 station.iStepAuto:= 120;
	120:
					arTonDelay[03](IN:= TRUE , PT:=T#50MS , Q=> , ET=> );
					IF arTonDelay[03].Q THEN
						 station.iStepAuto:=130;
				 			arTonDelay[03](IN:=FALSE, PT:=T#50MS , Q=> , ET=> );
				   END_IF
	130:
					fbROTAxisMove.xMoveAuto[2]:=TRUE;
				 IF fbROTAxisMove.xMoveInPos[2] THEN
					 station.iStepAuto :=140; 
				 END_IF	
	140://计算链条移动次数
				tsModuleProcess[1].xProcessCompleted:=TRUE;
				bCounter:=bCounter +1;
				station.iStepAuto:=142;	
	142://是否需要回原点
			  IF 	bCounter >8 THEN
						station.iStepAuto:=1000;	
				ELSE
				 			station.iStepAuto:=150;	
				END_IF
	150://数据传递
			FOR i:=4 TO 1 BY -1 DO
						MEMCPY(ADR(arBeltLineFixtureData[i+2]),ADR(arBeltLineFixtureData[i]),SIZEOF(arBeltLineFixtureData[i]));
			END_FOR
			 station.iStepAuto:=160;
	160://启动各个工位
			fbStation[7].xDone:=FALSE;
			fbStation[9].xDone:=FALSE;
			station.iStepAuto:=500;	
	500://清除本站过程记录
			FOR i:=1 TO gc_ModuleProNo BY 1 DO
				MEMSET(ADR(tsModuleProcess[i]),0,SIZEOF(tsModuleProcess[i]));
			END_FOR
			 station.iStepAuto:=999;
			
	999://----Single Run Finish----
		station.iStepAuto :=0;
		IF NOT station.xSingleContinuousRun THEN
			station.xSingleRunFlag:=FALSE;
		END_IF
		station.xCycleEnable:=FALSE;	
		station.xDone:=TRUE;	

1000://回原点流程
				fbROTAxisMove.xReferenceAuto := TRUE ;
				station.iStepAuto:=1010;	
1010://伺服回原点完成
	IF  fbAxisHome[16].home_done THEN 
		 fbROTAxisMove.xReferenceAuto  := FALSE ;
		 	station.iStepAuto:=1050;	
	END_IF
//1020://如果有报警
//		IF		fbROTAxisMove.xError THEN
//		 		fbROTAxisMove.xAlarmResetHmi:=TRUE;
//		ELSE
//		 		fbROTAxisMove.xAlarmResetHmi:=FALSE;	
//				 station.iStepAuto:=1050;	  
//		END_IF
1050://回原点完成
				tsModuleProcess[2].xProcessCompleted:=TRUE;
				_xFirstCycle:=FALSE;
				bCounter:=1;	
				station.iStepAuto:=142;	
				


	
	ELSE
		;	
END_CASE
END_IF
END_ACTION

ACTION FlowInit:
IF NOT station.xIniting THEN
  station.iStepInit:=0;    
ELSE
//--------------------------------------------初始化步序----------------------------------
CASE station.iStepInit OF	
 0://  
  	IF station.xIniting THEN	
  	  station.iStepInit:=10;	
  	END_IF	
10://复位数据
	bCounter:=1;
	_xFirstCycle:=FALSE;
	station.iStepInit:=20;
20://伺服上电
	fbROTAxisMove.xPowerInit :=TRUE;
	IF  fbROTAxisMove.xPowerOn THEN
			station.iStepInit:=30;
	END_IF
30: //伺服回原点
	fbROTAxisMove.xReferenceAuto := TRUE ;
	station.iStepInit:=40;
40://伺服回原点完成
	IF  fbAxisHome[16].home_done THEN 
		 fbROTAxisMove.xReferenceAuto  := FALSE ;
		 station.iStepInit:=50;  
	END_IF
50: //再次伺服回原点，保证位置
	fbROTAxisMove.xReferenceAuto := TRUE ;
	station.iStepInit:=60;
60://伺服回原点完成
	IF  fbAxisHome[16].home_done THEN 
		 fbROTAxisMove.xReferenceAuto  := FALSE ;
		 station.iStepInit:=70;  
	END_IF	
//65://如果有报警
//		IF		fbROTAxisMove.xError THEN
//		 		fbROTAxisMove.xAlarmResetHmi:=TRUE;
//		ELSE
//		 		fbROTAxisMove.xAlarmResetHmi:=FALSE;	
//				 station.iStepInit:=70;  
//		END_IF
70://伺服去待机点
	fbROTAxisMove.xMoveAuto[1]:=TRUE;
	IF  fbROTAxisMove.xMoveInPos[1] THEN
		 station.iStepInit:=999; 
	END_IF
999://初始化完成	
	station.iStepInit:=0;
	station.xInitDone:=TRUE;  
END_CASE
END_IF
END_ACTION

ACTION General:
{region "计算环形线周长程序"}
CASE wActionCalibration OF   
  10://回原点
  fbROTAxisMove.xReferenceAuto:= TRUE ;
  	wActionCalibration:=15;
  15:
	 IF  fbAxisHome[16].home_done THEN 
		 fbROTAxisMove.xReferenceAuto  := FALSE ;
		wActionCalibration:=100;
	 END_IF
  20://Jog正向，遇到原点传感器停止
   stData.Axis[16].rJogVelocity :=0.1;  
	fbROTAxisMove.xJogForwardAuto := TRUE ;
	 IF  arAxisSensorH[16] THEN 
		 fbROTAxisMove.xJogForwardAuto := FALSE ; 
			wActionCalibration:=30;
			rStartPoition[t]:=fbROTAxisMove.rActPos;
	 END_IF 
  60: //高速走定位，理论值前10MM处停止
	stData.Axis[16].rMovePosition[5] :=(755*5)-10; 
	wActionCalibration:=70;
	
70:
	fbROTAxisMove.xMoveAuto[5] := TRUE ;
	 IF fbROTAxisMove.xMoveInPos[5] THEN 
	 fbROTAxisMove.xMoveAuto[5] := FALSE ; 
	 wActionCalibration:=80;
	 END_IF 
80:
	  stData.Axis[16].rJogVelocity :=0.1;  
	fbROTAxisMove.xJogForwardAuto := TRUE ;
 IF   arAxisSensorH[16] THEN 
	 fbROTAxisMove.xJogForwardAuto := FALSE ; 
 		wActionCalibration:=90;
		rEndPoition[t]:=fbROTAxisMove.rActPos;
 END_IF 
90:
		stData.Axis[16].rRelativeDistance:=((rEndPoition[t]-rStartPoition[t])/85);
		wActionCalibration:=0;
END_CASE  
  
{endregion}
	 
{region "去下一个位置"}
NextPosR_TRIG(CLK:= fbMachine[1].xManualMode AND fbROTAxisMove.xMoveHmi[6], Q=> );
IF  NextPosR_TRIG.Q THEN
 stData.Axis[16].rMovePosition[6]:=fbROTAxisMove.rActPos +fbROTAxisMove.rRelativeDistance;
END_IF
  
{endregion}
END_ACTION

ACTION ILC:

//---------------------------------------------------工站可执行-------------------------------------------------------
station.xCanRun :=TRUE ;

//---------------------------------------------------气缸动作条件-------------------------------------------



//---------------------------------------------------伺服动作条件-------------------------------------------



fbROTAxisMove.xRunILC := 
fbROTAxisMove.xMoveILC[1] :=
fbROTAxisMove.xMoveILC[2] :=
fbROTAxisMove.xMoveILC[3] :=
fbROTAxisMove.xMoveILC[4] :=
fbROTAxisMove.xMoveILC[5] := TRUE ;
fbROTAxisMove.xRelativeILC:=TRUE;
END_ACTION

ACTION TipAuto:

//------------------------------------------------AutoTip Cylinder--------------------------------
//------------------------------------------------AutoTip Servo--------------------------------
//**************************************
//FOR i:= 1 TO 5 BY 1 DO 
//	IF fbROTAxisMove.xMoveAuto[i] THEN
//		fbROTAxisMove.iPosNumber := i ;
//	END_IF
//	
//END_FOR
//
//
//IF  fbMachine[1].xAutoMode AND NOT fbMachine[1].xRunning AND arTonDelay[10].Q   THEN
//	IF	fbROTAxisMove.iPosNumber=1 	AND NOT fbROTAxisMove.xMoveInPos[1] 	THEN 	station.adwAutoTip[1].10:=TRUE	;	END_IF//轴伺服自动时位置不在位置1
//	if	fbROTAxisMove.iPosNumber=2	AND NOT fbROTAxisMove.xMoveInPos[2]	THEN 	station.adwAutoTip[1].11:=TRUE	;	END_IF//轴伺服自动时位置不在位置2
//	if	fbROTAxisMove.iPosNumber=3	AND NOT fbROTAxisMove.xMoveInPos[3]	THEN 	station.adwAutoTip[1].12:=TRUE	;	END_IF//轴伺服自动时位置不在位置3
//	if	fbROTAxisMove.iPosNumber=4	AND NOT fbROTAxisMove.xMoveInPos[4]	THEN 	station.adwAutoTip[1].13:=TRUE	;	END_IF//轴伺服自动时位置不在位置4
//	IF	fbROTAxisMove.iPosNumber=5	AND NOT fbROTAxisMove.xMoveInPos[5]	THEN 	station.adwAutoTip[1].14:=TRUE	;	END_IF//轴伺服自动时位置不在位置5
//END_IF
END_ACTION

ACTION TipManual:
//--------------------------------------------ManualTip------------------------------------------------------

//-------------------------------------------气缸提示---------------------------------------------------------




/////////////////////////////////////////////////////////////////////////////////////////////////////////////////
END_ACTION

ACTION Z_Output:
(**************************气缸输出********************************)
END_ACTION

END_PROGRAM

// ---- POUs/001_Station/S09_CardCarrying.TcPOU
PROGRAM S09_CardCarrying
VAR
	//工站
	station					: REFERENCE TO FB_Station:=fbstation[9];
	//气缸
	fbHOZCyl	:REFERENCE TO FB_Cylinder:=fbCylinder[33];	//	卡片上料Y轴气缸
	fbVTCCyl_1	:REFERENCE TO FB_Cylinder:=fbCylinder[34];	//	卡片上料Z轴气缸1(上)
	fbVTCCyl_2	:REFERENCE TO FB_Cylinder:=fbCylinder[35];	//	卡片上料Z轴气缸2（下）



	//伺服
	fbZAxisStepMotor1	 :REFERENCE TO FB_Axis:=fbAxis[17];	//	卡片顶升步进
	fbZAxisStepMotor2	 :REFERENCE TO FB_Axis:=fbAxis[18];	//	卡片顶升步进
	//离子风棒
	Cimcor	 :REFERENCE TO FB_Cimcor_IZN10E:=fbCimcor[1];	//卡片离子风棒

	//延时
	arTonDelay :ARRAY[1..20] OF TON;
	//返回值
	UdiReturnValue :ARRAY[1..20] OF UDINT;
	//过程记录
	tsModuleProcess:ARRAY[1..gc_ModuleProNo] OF DUT_Process;
	xClearModuleProcessDone:BOOL;
	bClearProcessStep	:BYTE;
	i: INT;
	
	// //破真空
	arxVacuum_BreakValveControl:ARRAY[1..2]OF BOOL;
	// //破真空完成
	arxVacuum_BreakCompleted:ARRAY[1..2] OF BOOL;
	// //卡片到位传感器
	arxCardSensorReached: ARRAY[1..2] OF BOOL;
	// //卡片存在检测
	arxCardCheckSensor: ARRAY[1..2] OF BOOL;
	
	 //报警屏蔽
	_AlarmDisable: BOOL;
	// //真空吸动作
	arxVacuum_WorkValveControl: ARRAY[1..2] OF BOOL;
	// //真空吸到达真空
	arxVacuumWorkCompleted:ARRAY[1..2] OF BOOL;
	// //皮带线上检测卡片
	xBeltCardCheckSensor:ARRAY[1..2] OF BOOL;
	// //允许机械手放置深孔板
	xPutBoxPermit: BOOL;
	//首次循环
	_FirstCycle: ARRAY[1..10]OF BOOL;
	arxVacuum1_FeedValveWork: Array[1..2] of BOOL;
	arxVacuum1_FeedValveBroken: ARRAY[1..2] of bool;
	arxVacuumControlSensor: ARRAY[1..2] of BOOL;
	arxBrokenVacuumSensor: ARRAY[1..2] of BOOL;
	VacuumR_TRIG: ARRAY[1..2] of R_TRIG;
	VacuumBrokenR_TRIG: ARRAY[1..2] OF R_TRIG;
	arxAxisDone:ARRAY[1..2] OF BOOL;
END_VAR

A_Input();
Alarm();
Delay();
FlowAuto();
FlowInit();
General();
ILC();
TipAuto();
TipManual();
Z_Output();

ACTION A_Input:
//气缸
fbHOZCyl.xWP_Sensor	:=	IxS08HOZCylWP	;
fbHOZCyl.xHP_Sensor	:=	IxS08HOZCylHP	;
fbVTCCyl_1.xWP_Sensor	:=	IxS08VTCCyl_1WP	;
fbVTCCyl_1.xHP_Sensor	:=	IxS08VTCCyl_1HP	;
fbVTCCyl_2.xWP_Sensor	:=	IxS08VTCCyl_2WP	;
fbVTCCyl_2.xHP_Sensor	:=	IxS08VTCCyl_2HP	;
//传感器
xBeltCardCheckSensor[1]:= IxBeltEntryCardCheckSensor1;
xBeltCardCheckSensor[2]:= IxBeltEntryCardCheckSensor2;

//卡片检测
arxCardCheckSensor[1] := IxS08CardChcekSensor1;//	卡片工位¶有无传感器1
arxCardCheckSensor[2] :=  IxS08CardChcekSensor2;//	卡片工位¶有无传感器2

arxCardSensorReached[1] := NOT IxS08CardSensor1Reached	;//	卡片工位¶产品到位传感器1
arxCardSensorReached[2] := NOT  IxS08CardSensor2Reached	;//	卡片工位¶产品到位传感器2
END_ACTION

ACTION Alarm:
//
station.adwAlarm[1].00:=station.xInitTimeout;	  			//S09CardCarrying 初始化超时
//station.adwAlarm[1].01:=TRUE;	  							//S09CardCarrying 卡片不足，需要补充
station.adwAlarm[1].02:=Cimcor.xQError;	  		//S09CardCarrying 卡片离子风棒动作超时，请检查
station.adwAlarm[1].03:=Cimcor.xQNeedMaint;	  		//S09CardCarrying 卡片离子风棒需要维护，请检查
END_ACTION

ACTION Delay:
arTonDelay[01](IN:= , PT:=T#0.1S , Q=> , ET=> );
//arTonDelay[02](IN:=  , PT:=T#1S , Q=> , ET=> );//已被使用
arTonDelay[03](IN:=   , PT:=T#1S , Q=> , ET=> );
arTonDelay[04](IN:= , PT:=T#0.1S , Q=> , ET=> );
arTonDelay[05](IN:= , PT:=T#0.1S , Q=> , ET=> );
arTonDelay[06](IN:= , PT:=T#0.1S , Q=> , ET=> );
arTonDelay[07](IN:= , PT:=T#0.1S , Q=> , ET=> );
arTonDelay[08](IN:= , PT:=T#0.1S , Q=> , ET=> );
arTonDelay[09](IN:=NOT fbZAxisStepMotor1.xbusy  , PT:=T#0.1S , Q=> , ET=> );//TipAuto使用
arTonDelay[10](IN:= NOT  fbZAxisStepMotor2.xbusy , PT:=T#0.1S , Q=> , ET=> );//TipAuto使用
END_ACTION

ACTION FlowAuto:

//-----------------------------------------初始化是否完成判断----------------------------------------------
IF NOT station.xInitDone 
THEN
 	station.iStepAuto:=0;
 	station.xDone:=FALSE;
ELSIF station.xRunning  OR
 (tsModuleProcess[1].xProcessStarted AND NOT tsModuleProcess[1].xProcessCompleted) OR//卡片步进JOG
 (tsModuleProcess[2].xProcessStarted AND NOT tsModuleProcess[2].xProcessCompleted) 
THEN
//-----------------------------------------动作步骤--------------------------------------------------------
CASE station.iStepAuto OF	  
	0: //----Home Step，等待启动----
		IF station.xDisabled 
			AND station.xCanRun 
			AND NOT fbMachine[1].xStopped 
			AND NOT station.xSingleRunning 
		THEN
			station.xDone:=TRUE;
		END_IF
		
		IF  station.xSingleRunning 
			OR station.xCanRun 
			//AND NOT station.xDone 
			AND NOT station.xDisabled 
			AND NOT fbMachine[1].xStopped
		THEN
			station.xCycleEnable:=TRUE;
			//station.xDone:= FALSE;  
			station.iStepAuto:= 10;
		END_IF
  10: //复位数据 
			fbZAxisStepMotor1.xJogForwardAuto:=FALSE;
			fbZAxisStepMotor2.xJogForwardAuto:=FALSE;
			fbZAxisStepMotor1.xJogForwardHMI:=FALSE;
			fbZAxisStepMotor2.xJogForwardHMI:=FALSE;
			IF  station.xSingleRunning THEN
				 FOR i:=1 TO gc_ModuleProNo BY 1 DO
						 MEMSET(ADR(tsModuleProcess[i]),0,SIZEOF(tsModuleProcess[i]));
				 END_FOR
			END_IF
			station.iStepAuto:=20;	
	20://检查卡片是否在位
			_AlarmDisable:=FALSE;
			IF arxCardCheckSensor[1] AND
				arxCardCheckSensor[2] THEN
				station.iStepAuto:=30;
 			ELSE
				station.iStepAuto:=25;
			END_IF
	25://卡片缺少,伺服回参考点
			 fbZAxisStepMotor1.xMoveAuto[1]:=TRUE;
			 fbZAxisStepMotor2.xMoveAuto[1]:=TRUE;
			IF    fbZAxisStepMotor1.xMoveInPos[1] AND 
				fbZAxisStepMotor2.xMoveInPos[1] THEN
				station.iStepAuto:=26;
			END_IF
	26://卡片确实报警
			IF NOT  _AlarmDisable  THEN
				station.adwAlarm[1].01:=TRUE;//S09CardCarrying 卡片不足，需要补充
				_AlarmDisable:=TRUE;
			END_IF
				station.iStepAuto:=20;
	30://步进JOG流程开始
			tsModuleProcess[1].xProcessNotStarted:=TRUE;
			stData.Axis[17].rJogVelocity :=5;  
			stData.Axis[18].rJogVelocity :=5;  
			station.iStepAuto:=31;
	31://步进上升等待到达传感器
			tsModuleProcess[1].xProcessStarted:=TRUE;
			IF  NOT station.xSingleRunning THEN 
					IF 	NOT arxCardSensorReached[1]  THEN
						fbZAxisStepMotor1.xJogForwardAuto:=TRUE;
					ELSE
						fbZAxisStepMotor1.xJogForwardAuto:=FALSE;
					END_IF
					IF 	NOT 	arxCardSensorReached[2]  THEN
						fbZAxisStepMotor2.xJogForwardAuto:=TRUE;
					ELSE
						fbZAxisStepMotor2.xJogForwardAuto:=FALSE;
					END_IF
			ELSE
			 		IF 	NOT arxCardSensorReached[1]   THEN
						fbZAxisStepMotor1.xJogForwardHmi:=TRUE;
					ELSE
						fbZAxisStepMotor1.xJogForwardHmi:=FALSE;
					END_IF
					IF 	NOT 	arxCardSensorReached[2]   THEN
						fbZAxisStepMotor2.xJogForwardHmi:=TRUE;
					ELSE
						fbZAxisStepMotor2.xJogForwardHmi:=FALSE;
					END_IF
			END_IF
			IF  arxCardSensorReached[1]  AND 
				arxCardSensorReached[2]  THEN
				station.iStepAuto:=35;
			END_IF
	35://步进JOG流程完成,离子风棒启动
		tsModuleProcess[1].xProcessCompleted:=TRUE;
			Cimcor.xIStart:=TRUE;
			station.iStepAuto:=40;
	40://X轴气缸伸出
		fbHOZCyl.xAuto :=TRUE;
		IF fbHOZCyl.xWP_Delay THEN
			station.iStepAuto:=50;
		END_IF
	50://上Z轴下降
		fbVTCCyl_1.xAuto:=TRUE;
		IF fbVTCCyl_1.xWP_Delay THEN
			station.iStepAuto:=60;	
		END_IF
	60://下Z轴下降
		arTonDelay[02](IN:=FALSE); 
		fbVTCCyl_2.xAuto:=TRUE;
		IF fbVTCCyl_2.xWP_Delay THEN
			station.iStepAuto:=90;	
		END_IF
	90://真空吸动作
			arTonDelay[02](IN:=TRUE  , PT:=T#5S , Q=> , ET=> );
			fbSmcVacuum[1].xIVacuumWork:=TRUE;
			fbSmcVacuum[2].xIVacuumWork:=TRUE;
			IF  fbSmcVacuum[1].xIVacuumWorkReached AND 
			 		fbSmcVacuum[2].xIVacuumWorkReached THEN
						station.iStepAuto:= 100;
			ELSIF arTonDelay[02].Q THEN
			 			station.iStepAuto:= 100;//动作超时也放行
						arTonDelay[02](IN:=FALSE);
			END_IF
	100://真空吸动作完成
			station.iStepAuto:= 110;
	110://上Z轴上升
			fbVTCCyl_1.xAuto:=FALSE;
		IF fbVTCCyl_1.xHP_Delay THEN
			station.iStepAuto:=120;	
		END_IF
	120://
				station.iStepAuto:= 130;
				
	130://	开始抖动流程
				fbVTCCyl_2.xAuto:=FALSE;
				IF fbVTCCyl_2.xHP_Delay THEN
					station.iStepAuto:=140;	
				END_IF	
	140:		
				fbVTCCyl_2.xAuto:=TRUE;
				IF fbVTCCyl_2.xWP_Delay THEN
					station.iStepAuto:=150;	
				END_IF		
	150://抖动完成
			station.iStepAuto:=160;		
	160://下Z轴上升
				fbVTCCyl_2.xAuto:=FALSE;
				IF fbVTCCyl_2.xHP_Delay THEN
					station.iStepAuto:=161;	
				END_IF	
	161://检测卡片时是否还在	
				IF NOT  fbSmcVacuum[1].xIVacuumWorkReached OR 
			 		 NOT fbSmcVacuum[2].xIVacuumWorkReached THEN
							fbSmcVacuum[1].xIVacuumBroken:=TRUE;
								fbSmcVacuum[2].xIVacuumBroken:=TRUE;
						IF  fbSmcVacuum[1].xIVacuumBrokenReached AND 
								fbSmcVacuum[2].xIVacuumBrokenReached THEN
										station.iStepAuto:=40;//重新去取卡片	
						END_IF
				ELSE
									station.iStepAuto:=165;
				END_IF
	165://检查是否允许放卡片
					Cimcor.xIStop:=TRUE;
			 IF   NOT   station.xSingleRunning THEN 
					 IF  NOT xBeltCardCheckSensor[1] AND 
						 NOT xBeltCardCheckSensor[2] AND 
						 NOT  station.xdone 			AND
						 (NOT _FirstCycle[1] OR S10_BeltCarrying.station.xDone )THEN 
						 station.iStepAuto:=180;
						 _FirstCycle[1]:=TRUE;
					 END_IF
			 ELSE
					 station.iStepAuto:=180;
			 END_IF
	180:
				station.iStepAuto:= 190;
	190://Y轴回原点
				fbHOZCyl.xAuto:=FALSE;
				IF fbHOZCyl.xHP_Delay THEN
					station.iStepAuto:=200;	
				END_IF		
	200://上Z轴气缸下降
				fbVTCCyl_1.xAuto:=TRUE;
				IF fbVTCCyl_1.xWP_Delay THEN
					station.iStepAuto:=220;	
				END_IF							
	220://下Z轴气缸下降
				fbVTCCyl_2.xAuto:=TRUE;
				IF fbVTCCyl_2.xWP_Delay THEN
					station.iStepAuto:=230;	
				END_IF			
	230://破真空
				fbSmcVacuum[1].xIVacuumBroken:=TRUE;
				fbSmcVacuum[2].xIVacuumBroken:=TRUE;
				IF  fbSmcVacuum[1].xIVacuumBrokenReached AND 
				 		fbSmcVacuum[2].xIVacuumBrokenReached THEN
				 station.iStepAuto:=240;		
				END_IF
	240://流程完成
				 station.iStepAuto:=250;
	250://上Z轴上升
				fbVTCCyl_1.xAuto:=FALSE;
				IF fbVTCCyl_1.xHP_Delay THEN
					station.iStepAuto:=260;	
				END_IF
	260://下Z轴上升
				fbVTCCyl_2.xAuto:=FALSE;
				IF fbVTCCyl_2.xHP_Delay THEN
					station.iStepAuto:=270;	
				END_IF
	270://检查卡片检测是否在位
		IF  xBeltCardCheckSensor[1] AND 
			xBeltCardCheckSensor[2] THEN
			 station.iStepAuto:=280;
		END_IF
	280://已放入卡片
			arBeltLineFixtureData[1].xMaterialOnOff:=TRUE;
			arBeltLineFixtureData[2].xMaterialOnOff:=TRUE;
			arBeltLineFixtureData[1].stProduct.xCardLoading_OK:=TRUE;
			arBeltLineFixtureData[1].stProduct.xCardLoading_NOK:=FALSE;
			arBeltLineFixtureData[2].stProduct.xCardLoading_OK:=TRUE;
			arBeltLineFixtureData[2].stProduct.xCardLoading_NOK:=FALSE;
			station.iStepAuto:=300;
	290://未放入卡片
			arBeltLineFixtureData[1].xMaterialOnOff:=FALSE;
			arBeltLineFixtureData[2].xMaterialOnOff:=FALSE;
			arBeltLineFixtureData[1].stProduct.xCardLoading_OK:=FALSE;
			arBeltLineFixtureData[1].stProduct.xCardLoading_NOK:=FALSE;
			arBeltLineFixtureData[2].stProduct.xCardLoading_OK:=FALSE;
			arBeltLineFixtureData[2].stProduct.xCardLoading_NOK:=FALSE;
			station.iStepAuto:=300;
	300://清除过程数据
			FOR i:=1 TO gc_ModuleProNo BY 1 DO
				MEMSET(ADR(tsModuleProcess[i]),0,SIZEOF(tsModuleProcess[i]));
			END_FOR
			station.iStepAuto:=999;
			
	999://----Single Run Finish----
			
		station.iStepAuto :=0;
		IF NOT station.xSingleContinuousRun THEN
			station.xSingleRunFlag:=FALSE;
		END_IF
		
		station.xCycleEnable:=FALSE;	
		station.xDone:=TRUE;
	ELSE
		;	
END_CASE


END_IF
END_ACTION

ACTION FlowInit:
IF NOT station.xIniting THEN
  station.iStepInit:=0;    
ELSE
//--------------------------------------------初始化步序----------------------------------
CASE station.iStepInit OF	
 0://  
  	IF station.xIniting THEN	
  	  station.iStepInit:=10;	
  	END_IF	
10://复位数据
			Cimcor.xIReset:=TRUE;
			fbZAxisStepMotor1.xJogForwardAuto:=FALSE;
			fbZAxisStepMotor2.xJogForwardAuto:=FALSE;
			fbZAxisStepMotor1.xJogForwardHMI:=FALSE;
			fbZAxisStepMotor2.xJogForwardHMI:=FALSE;
			fbZAxisStepMotor1.xJogBackwardsHmi:=FALSE;
			fbZAxisStepMotor2.xJogBackwardsHmi:=FALSE;
			station.iStepInit:=30;
//20://检查是否需要破真空	
//	IF tsModuleProcess[1].xProcessStarted AND
//		 NOT tsModuleProcess[1].xProcessCompleted THEN
//		 station.iStepInit:=30;
//	ELSE
//		station.iStepInit:=40;	
//	END_IF
30://破真空
			fbSmcVacuum[1].xIVacuumBroken:=TRUE;
			fbSmcVacuum[2].xIVacuumBroken:=TRUE;
				station.iStepInit:=35;	
35://真空已破
		IF  fbSmcVacuum[1].xIVacuumBrokenReached AND 
				 fbSmcVacuum[2].xIVacuumBrokenReached THEN
				station.iStepInit:=40;	
				END_IF
40://上Z轴上升
	fbVTCCyl_1.xInit:=TRUE;
	IF  fbVTCCyl_1.xHP_Delay THEN
		station.iStepInit:=50;	
	END_IF
50://下轴上升
	fbVTCCyl_2.xInit:=TRUE;
	IF  fbVTCCyl_2.xHP_Delay THEN
		station.iStepInit:=60;	
	END_IF
60://X轴气缸回原
	fbHOZCyl.xInit:=TRUE;
	IF  fbHOZCyl.xHP_Delay THEN
		station.iStepInit:=65;	
	END_IF		
65://卡片步进上电
	fbZAxisStepMotor1.xPowerInit:=TRUE;
	fbZAxisStepMotor2.xPowerInit:=TRUE;
	IF		fbZAxisStepMotor1.xPowerOn AND
		    fbZAxisStepMotor2.xPowerOn THEN
			station.iStepInit:=70;	
	END_IF
70://卡片1步进
			IF NOT  arxCardCheckSensor[2] THEN
					 IF  NOT  arAxisSensorH[18] THEN
									 fbZAxisStepMotor2.xJogBackwardsHmi:=TRUE;
						ELSE		
						 			fbZAxisStepMotor2.xJogBackwardsHmi:=FALSE;
									arxAxisDone[1]:=TRUE;	
						END_IF
						
			ELSE
					arxAxisDone[1]:=TRUE;	
			END_IF
	 	//卡片2步进
			 IF NOT  arxCardCheckSensor[1] THEN
						IF  NOT  arAxisSensorH[17] THEN
										fbZAxisStepMotor1.xJogBackwardsHmi:=TRUE;
						 ELSE		
									 fbZAxisStepMotor1.xJogBackwardsHmi:=FALSE;
									 	arxAxisDone[2]:=TRUE;	
						 END_IF
			 ELSE
					  	arxAxisDone[2]:=TRUE;	
			 END_IF
		//判断是否完成
			IF  arxAxisDone[1] AND 
			 		arxAxisDone[2] THEN
					station.iStepInit:=999;	
			END_IF
//80://回原点
//	fbZAxisStepMotor1.xReferenceAuto:=TRUE;
//	fbZAxisStepMotor2.xReferenceAuto:=TRUE;
//	station.iStepinit:=90;
//90:
//   IF  fbAxisHome[17].home_done  AND 
//		fbAxisHome[18].home_done THEN 
//		fbZAxisStepMotor1.xAlarmResetHmi:=TRUE;
//		fbZAxisStepMotor2.xAlarmResetHmi:=TRUE;
//		 fbZAxisStepMotor1.xReferenceAuto:=FALSE;
//		fbZAxisStepMotor2.xReferenceAuto:=FALSE;
//		 station.iStepInit:=100;  
//	END_IF

//100://参考点
//			 fbZAxisStepMotor1.xMoveAuto[1]:=TRUE;
//			 fbZAxisStepMotor2.xMoveAuto[1]:=TRUE;
//			IF    fbZAxisStepMotor1.xMoveInPos[1] AND 
//				fbZAxisStepMotor2.xMoveInPos[1] THEN
//				station.iStepInit:=999;
//			END_IF
999://初始化完成	
	station.iStepInit:=0;
	station.xInitDone:=TRUE;  
END_CASE
END_IF
END_ACTION

ACTION General:

END_ACTION

ACTION ILC:

//---------------------------------------------------工站可执行-------------------------------------------------------
station.xCanRun :=TRUE ;

//---------------------------------------------------气缸动作条件-------------------------------------------

fbHOZCyl.xOffILC	:=	TRUE;//fbVTCCyl_1.xHP_Delay AND  fbVTCCyl_1.xHP_Delay 	;
fbHOZCyl.xOnILC		:=	TRUE;//fbVTCCyl_1.xHP_Delay AND  fbVTCCyl_1.xHP_Delay	;
fbVTCCyl_1.xOffILC	:=	TRUE;//fbHOZCyl.xHP_Delay OR fbHOZCyl.xWP_Delay	;
fbVTCCyl_1.xOnILC	:=	TRUE;//fbHOZCyl.xHP_Delay OR fbHOZCyl.xWP_Delay	;
fbVTCCyl_2.xOffILC	:=	TRUE	;
fbVTCCyl_2.xOnILC	:=	TRUE; //fbHOZCyl.xHP_Delay OR fbHOZCyl.xWP_Delay	;


//---------------------------------------------------伺服动作条件-------------------------------------------


fbZAxisStepMotor1.xRunILC := 
fbZAxisStepMotor1.xMoveILC[1] :=
fbZAxisStepMotor1.xMoveILC[2] :=
fbZAxisStepMotor1.xMoveILC[3] :=
fbZAxisStepMotor1.xMoveILC[4] :=
fbZAxisStepMotor1.xMoveILC[5] := TRUE ;


fbZAxisStepMotor2.xRunILC := 
fbZAxisStepMotor2.xMoveILC[1] :=
fbZAxisStepMotor2.xMoveILC[2] :=
fbZAxisStepMotor2.xMoveILC[3] :=
fbZAxisStepMotor2.xMoveILC[4] :=
fbZAxisStepMotor2.xMoveILC[5] := TRUE ;



fbSmcVacuum[1].xIDeviceRunning:=TRUE;
fbSmcVacuum[2].xIDeviceRunning:=TRUE;
END_ACTION

ACTION TipAuto:

//------------------------------------------------AutoTip Cylinder--------------------------------
station.adwAutoTip[1].00	:=	fbHOZCyl.xAutoTip	;
station.adwAutoTip[1].01	:=	fbVTCCyl_1.xAutoTip	;
station.adwAutoTip[1].02	:=	fbVTCCyl_2.xAutoTip	;	
//------------------------------------------------AutoTip Servo--------------------------------
//**************************************
//FOR i:= 1 TO 5 BY 1 DO 
//	IF fbZAxisStepMotor1.xMoveAuto[i] THEN
//		fbZAxisStepMotor1.iPosNumber := i ;
//	END_IF
//	IF fbZAxisStepMotor2.xMoveAuto[i] THEN
//		fbZAxisStepMotor2.iPosNumber := i ;
//	END_IF
//	
//END_FOR
//
//
//IF  fbMachine[1].xAutoMode AND NOT fbMachine[1].xRunning AND arTonDelay[09].Q THEN
//	IF	fbZAxisStepMotor1.iPosNumber=1 	AND NOT fbZAxisStepMotor1.xMoveInPos[1] 	THEN 	station.adwAutoTip[1].15:=TRUE	;	END_IF//轴伺服自动时位置不在位置1
//	if	fbZAxisStepMotor1.iPosNumber=2	AND NOT fbZAxisStepMotor1.xMoveInPos[2]	THEN 	station.adwAutoTip[1].16:=TRUE	;	END_IF//轴伺服自动时位置不在位置2
//	if	fbZAxisStepMotor1.iPosNumber=3	AND NOT fbZAxisStepMotor1.xMoveInPos[3]	THEN 	station.adwAutoTip[1].17:=TRUE	;	END_IF//轴伺服自动时位置不在位置3
//	if	fbZAxisStepMotor1.iPosNumber=4	AND NOT fbZAxisStepMotor1.xMoveInPos[4]	THEN 	station.adwAutoTip[1].18:=TRUE	;	END_IF//轴伺服自动时位置不在位置4
//	IF	fbZAxisStepMotor1.iPosNumber=5	AND NOT fbZAxisStepMotor1.xMoveInPos[5]	THEN 	station.adwAutoTip[1].19:=TRUE	;	END_IF//轴伺服自动时位置不在位置5
//END_IF
//IF  fbMachine[1].xAutoMode AND NOT fbMachine[1].xRunning AND arTonDelay[10].Q THEN
//	IF	fbZAxisStepMotor2.iPosNumber=1 	AND NOT fbZAxisStepMotor2.xMoveInPos[1] 	THEN 	station.adwAutoTip[1].20:=TRUE	;	END_IF//轴伺服自动时位置不在位置1
//	if	fbZAxisStepMotor2.iPosNumber=2	AND NOT fbZAxisStepMotor2.xMoveInPos[2]	THEN 	station.adwAutoTip[1].21:=TRUE	;	END_IF//轴伺服自动时位置不在位置2
//	if	fbZAxisStepMotor2.iPosNumber=3	AND NOT fbZAxisStepMotor2.xMoveInPos[3]	THEN 	station.adwAutoTip[1].22:=TRUE	;	END_IF//轴伺服自动时位置不在位置3
//	if	fbZAxisStepMotor2.iPosNumber=4	AND NOT fbZAxisStepMotor2.xMoveInPos[4]	THEN 	station.adwAutoTip[1].23:=TRUE	;	END_IF//轴伺服自动时位置不在位置4
//	if	fbZAxisStepMotor2.iPosNumber=5	AND NOT fbZAxisStepMotor2.xMoveInPos[5]	THEN 	station.adwAutoTip[1].24:=TRUE	;	END_IF//轴伺服自动时位置不在位置5
//END_IF
END_ACTION

ACTION TipManual:
//--------------------------------------------ManualTip------------------------------------------------------

//-------------------------------------------气缸提示---------------------------------------------------------




/////////////////////////////////////////////////////////////////////////////////////////////////////////////////
END_ACTION

ACTION Z_Output:
//气缸输出
QxS08HOZCylWP	:=	fbHOZCyl.xWP_Valve	;
QxS08HOZCylHP	:=	fbHOZCyl.xHP_Valve	;
QxS08VTCCyl_1WP	:=	fbVTCCyl_1.xWP_Valve	;
QxS08VTCCyl_1HP	:=	fbVTCCyl_1.xHP_Valve	;
QxS08VTCCyl_2WP	:=	fbVTCCyl_2.xWP_Valve	;
QxS08VTCCyl_2HP	:=	fbVTCCyl_2.xHP_Valve	;
END_ACTION

END_PROGRAM

// ---- POUs/003_FB/0011_Cimcor/FB_Cimcor_IZN10E.TcPOU
FUNCTION_BLOCK FB_Cimcor_IZN10E
(*
********************************************************************************
* Name: FB_Cimcor_IZN10E
*
* Author:  Automanh
* Version: 1.0.0
*
* Description:
*  Function block for SMC IZN10E-0106 Cimcor and blow Valve
*
* Remarks:
*
* Revisions:
*   1.0 -AutomanH build
*********************************************************************************)
VAR_INPUT
 xIStart  :BOOL;//离子风棒及电磁阀启动
 xIStop		:BOOL;//离子风棒停止
 xIReset	:BOOL;//复位信号
 xICimcorMaint:BOOL;//维护信号
 xIError	:BOOL;//异常信号
 xICimcorStarted:BOOL;//离子风棒放电开始
END_VAR
VAR_OUTPUT
 xQError:BOOL;
 xQCimcorStart:BOOL;//true-离子风棒放电  false-离子风棒停止放电
 xQCimcorReset:BOOL;//复位离子风棒
 xQValveStart:BOOL;//电磁阀打开
 xQNeedMaint :BOOL;//需要维护
END_VAR
VAR
 iStartStep,iOldStartStep:INT;
 iStopStep,iOldStopStep:INT;
 iResetStep,iOldResetStep:INT;
 OperR_TRIG:ARRAY[1..4]OF R_TRIG;
 tDelay:TON;
 tTimeOut:ARRAY[1..3] OF TON;
END_VAR

ACT_Start();
ACT_Stop();
ACT_Reset();
ACT_Error();
ACT_Maint();

ACTION ACT_Error:
tTimeOut[1](IN:=  iStartStep=iOldStartStep AND iOldStartStep <>0, PT:= T#5S, Q=> , ET=> );
tTimeOut[2](IN:=  iStopStep=iOldStopStep AND iOldStopStep <>0, PT:= T#5S, Q=> , ET=> );
tTimeOut[3](IN:=  iResetStep=iOldResetStep AND iOldResetStep <>0, PT:= T#5S, Q=> , ET=> );
IF  tTimeOut[1].Q OR tTimeOut[2].Q OR  tTimeOut[3].Q OR xIError THEN
		xQError:=TRUE;
END_IF
END_ACTION

ACTION ACT_Maint:
//维护信号
IF  xICimcorMaint THEN
 	xQNeedMaint:=TRUE;
END_IF
END_ACTION

ACTION ACT_Reset:
OperR_TRIG[3](CLK:=xIReset , Q=> );
CASE iResetStep OF
 0://等待启动
 		IF  OperR_TRIG[3].Q THEN
				xIStop:=FALSE;
				xIStart:=FALSE;
				xIReset:=FALSE;
				xQError:=FALSE;
				iStartStep:=0;
				iStopStep:=0;
				iResetStep:=0;
				iResetStep:=iResetStep+1;
		END_IF
 1://复位离子封棒
 		iOldResetStep:=iResetStep;
 		xQCimcorStart:=FALSE;
		xQCimcorReset:=TRUE;
		tDelay(IN:=FALSE);
		iResetStep:=iResetStep+1;
 2://延时
 			iOldResetStep:=iResetStep;
 			tDelay(IN:= TRUE , PT:= T#200MS, Q=> , ET=> );
		IF tDelay.Q THEN
		 	iResetStep:=iResetStep+1;
			tDelay(IN:=FALSE);
		END_IF
 3://关闭复位信号
 		iOldResetStep:=iResetStep;
 		xQCimcorReset:=FALSE;
		iResetStep:=iResetStep+1;
 4://结束
 		iResetStep:=0;
END_CASE
END_ACTION

ACTION ACT_Start:
OperR_TRIG[1](CLK:=xIStart , Q=> );
CASE iStartStep OF
 0://等待启动
 		IF  OperR_TRIG[1].Q THEN
				xIStop:=FALSE;
				xIStart:=FALSE;
				iStopStep:=0;
				iStartStep:=iStartStep+1;
		END_IF
 1://开启离子风棒
 		iOldStartStep:=iStartStep;
 		xQCimcorStart:=TRUE;
		iStartStep:=iStartStep+1;
 2://检查离子风棒是否开启
 		iOldStartStep:=iStartStep;
 		IF xICimcorStarted THEN
					iStartStep:=iStartStep+1; 
		END_IF
 3://打开电磁阀
 		iOldStartStep:=iStartStep;
 		xQValveStart:=TRUE;
			iStartStep:=iStartStep+1; 
 4://结束
 		iStartStep:=0;
END_CASE
END_ACTION

ACTION ACT_Stop:
OperR_TRIG[2](CLK:=xIStop , Q=> );
CASE iStopStep OF
 0://等待启动
 		IF  OperR_TRIG[2].Q THEN
				xIStop:=FALSE;
				xIStart:=FALSE;
				iStopStep:=0;
				iStopStep:=iStopStep+1;
		END_IF
 1://关闭离子风棒
 		iOldStopStep:=iStopStep;
 		xQCimcorStart:=FALSE;
		iStopStep:=iStopStep+1;
 2://检查离子风棒是否关闭
 		iOldStopStep:=iStopStep;
 		IF  NOT xICimcorStarted THEN
					iStopStep:=iStopStep+1; 
		END_IF
 3://关闭电磁阀
 			iOldStopStep:=iStopStep;
 			xQValveStart:=FALSE;
			iStopStep:=iStopStep+1; 
 4://结束
 			iStopStep:=0;
END_CASE
END_ACTION

END_FUNCTION_BLOCK

// ---- POUs/001_Station/S11_Packing.TcPOU
PROGRAM S11_Packing
VAR
 //工站
	station					: REFERENCE TO FB_Station:=fbstation[11];
	//200smart通讯
	Modbus_200Smart	: REFERENCE TO FB_Modbus_200Smart:=fbModbus_200Smart;
	// 设备停止延时
	tStopDelay:Tc2_Standard.TON;
END_VAR

FlowAuto();
FlowInit();
ILC();
Mapping();
General();

ACTION FlowAuto:

//-----------------------------------------初始化是否完成判断----------------------------------------------
IF NOT station.xInitDone 
THEN
 	station.iStepAuto:=0;
 	station.xDone:=FALSE;
ELSIF station.xRunning  OR station.xRunningOffProhibit
THEN
//-----------------------------------------动作步骤--------------------------------------------------------
CASE station.iStepAuto OF	  
	0: //----Home Step，等待启动----
		IF station.xDisabled 
			AND station.xCanRun 
			AND NOT fbMachine[1].xStopped 
			AND NOT station.xSingleRunning 
		THEN
			station.xDone:=TRUE;
		END_IF
		
		IF  station.xSingleRunning 
			OR station.xCanRun 
			//AND NOT station.xDone 
			AND NOT station.xDisabled 
			AND NOT fbMachine[1].xStopped
		THEN
			station.xCycleEnable:=TRUE;
			//station.xDone:= FALSE;  
			
			station.iStepAuto:= 10;
		END_IF
   10: //复位数据 
			station.iStepAuto :=20;
	 20:	
				IF  sModbus_200SMART.iTemperatureReached  =1 THEN 
						station.iStepAuto:= 999;
					END_IF
	999://----Single Run Finish----
			
		station.iStepAuto :=0;
		IF NOT station.xSingleContinuousRun THEN
			station.xSingleRunFlag:=FALSE;
		END_IF
		
		station.xCycleEnable:=FALSE;	
		(*station.xDone:=TRUE;*)
	ELSE
		;	
END_CASE
END_IF
END_ACTION

ACTION FlowInit:
IF NOT station.xIniting THEN
  station.iStepInit:=0;    
ELSE
//--------------------------------------------初始化步序----------------------------------
CASE station.iStepInit OF	
 0://  
  	IF station.xIniting THEN	
  	  station.iStepInit:=10;	
  	END_IF	
10://复位数据
  station.iStepInit:=999;	
	
//20://等待初始化完成
//	IF  sModbus_200SMART.iInitCompleted =1 THEN
//	 			station.iStepInit:=999;	
//	END_IF
999://初始化完成	
	station.iStepInit:=0;
	station.xInitDone:=TRUE;  
END_CASE
END_IF
END_ACTION

ACTION General:
{region "停止"}
tStopDelay(IN:= fbMachine[1].xManualMode, PT:=T#60S , Q=> , ET=> );
IF tStopDelay.Q THEN
		station.xRunningOffProhibit:=FALSE;
ELSIF  station.iStepAuto =10 THEN
		station.xRunningOffProhibit:=TRUE;
END_IF	 
{endregion}
END_ACTION

ACTION ILC:

//---------------------------------------------------工站可执行-------------------------------------------------------
station.xCanRun :=TRUE ;

//---------------------------------------------------气缸动作条件-------------------------------------------
END_ACTION

ACTION Mapping:
(**********配置*********)
Modbus_200Smart.stPara.strSlaveIP:='192.168.1.2';
Modbus_200Smart.stPara.iSlavePort:=502;
Modbus_200Smart.stPara.bySlaveID:=1;
END_ACTION

END_PROGRAM

// ---- POUs/003_FB/0001_200Smart/FB_Modbus_200Smart.TcPOU
FUNCTION_BLOCK FB_Modbus_200Smart
(*
********************************************************************************
* Name: FB_Modbus_200Smart
*
* Author:  AutomanH
* Version: 1.0.0
*
* Description:
*	Beckhoff CX5130 and SIEMENS 200SMART Modbus TCP Communication 
*
* Remarks:
*
* Revisions:
*   V1.0.0 -Automanh 2022.06.01
*********************************************************************************)
VAR_INPUT
	stPara       : ST_Sys_Para;//系统参数	
END_VAR
VAR_IN_OUT
	st_IOData: DUT_200SMART;
END_VAR
VAR
 {attribute 'tc_no_symbol'}
	_aRead_VAR: ARRAY[1..5] OF FB_MBReadRegs;
	{attribute 'tc_no_symbol'}
	_aWtirt_VAR: ARRAY[1..5] OF FB_MBWriteRegs;
	{attribute 'tc_no_symbol'}
	pSysTo200Smart :  ARRAY[1..12] OF WORD;//Cx5130 to 200smart 数据
	{attribute 'tc_no_symbol'}
	pSysFrom200Smart :ARRAY[1..12] OF WORD ;//Cx5130 from 200smart 数据
END_VAR

ACT_Connect();
ACT_Mapping();

ACTION ACT_Connect:
//读取200smart数据
_aRead_VAR[1](
	sIPAddr:= stPara.strSlaveIP, 
	nTCPPort:= stPara.iSlavePort, 
	nUnitID:= stPara.bySlaveID, 
	nQuantity:= 7, 
	nMBAddr:= 0, 
	cbLength:= 14,
	pDestAddr:= ADR(pSysFrom200Smart), 
	bExecute:= stSysPulse.xP10ms, 
	tTimeout:=T#1S , 
	bBusy=> , 
	bError=> , 
	nErrId=> , 
	cbRead=> );
	
//写入200smart数据
_aWtirt_VAR[1](
	sIPAddr:=stPara.strSlaveIP , 
	nTCPPort:=stPara.iSlavePort , 
	nUnitID:=stPara.bySlaveID , 
	nQuantity:= 5, 
	nMBAddr:= 11, 
	cbLength:= 10,
	pSrcAddr:= ADR(pSysTo200Smart), 
	bExecute:=stSysPulse.xP10ms ,  
	tTimeout:=T#1S , 
	bBusy=> , 
	bError=> , 
	nErrId=> );
END_ACTION

ACTION ACT_Mapping:
st_IOData.iAlive           :=pSysFrom200Smart[1];
st_IOData.iInitCompleted 	 :=pSysFrom200Smart[2];
st_IOData.iStatus        	 :=pSysFrom200Smart[3];
st_IOData.iResult       	 :=pSysFrom200Smart[4];
st_IOData.iError         	 :=pSysFrom200Smart[5];
st_IOData.iBeltEnterEnable :=pSysFrom200Smart[6];
st_IOData.iTemperatureReached:=pSysFrom200Smart[7];
st_IOData.iRev2         	 :=pSysFrom200Smart[8];
st_IOData.iRev3        		 :=pSysFrom200Smart[9];
st_IOData.iRev4         	  :=pSysFrom200Smart[10];
st_IOData.iRev5		        :=pSysFrom200Smart[11];
//
pSysTo200Smart[1]:=st_IOData.iMachineMode	;
pSysTo200Smart[2]:=st_IOData.iMachineIniting	;
pSysTo200Smart[3]:=st_IOData.iMachineStart	;
pSysTo200Smart[4]:=st_IOData.iMachineStop	;
pSysTo200Smart[5]:=st_IOData.iMachineEstop	;
pSysTo200Smart[6]:=st_IOData.iMachineDisable	;
pSysTo200Smart[7]:=st_IOData.iRev6;
pSysTo200Smart[8]:=st_IOData.iRev7	;
pSysTo200Smart[9]:=st_IOData.iRev8	;
pSysTo200Smart[10]:=st_IOData.iRev9	;
pSysTo200Smart[11]:=st_IOData.iRev10	;
pSysTo200Smart[12]:=st_IOData.iRev11	;
END_ACTION

END_FUNCTION_BLOCK

// ---- POUs/001_Station/S12_PreLine.TcPOU
PROGRAM S12_PreLine
VAR
 //工站
	station					: REFERENCE TO FB_Station:=fbstation[12];
	//变频器
	ATV12						: REFERENCE TO FB_ATV12:=fbATV12;
	// 支线电机启动
	xPreLineMoveStart: BOOL;
	// 支线电机停止
	xPreLineMoveStop: BOOL;
	MotorStartR_TRIG: R_TRIG;
	MotorStopR_TRIG: R_TRIG;
	//设备停止延时
	tStopDelay:Tc2_Standard.TON;
END_VAR

A_Input();
FlowAuto();
FlowInit();
ILC();
General();
Z_Output();

ACTION A_Input:
//变频器
END_ACTION

ACTION FlowAuto:

//-----------------------------------------初始化是否完成判断----------------------------------------------
IF NOT station.xInitDone 
THEN
 	station.iStepAuto:=0;
 	station.xDone:=FALSE;
ELSIF station.xRunning   OR station.xRunningOffProhibit  
THEN
//-----------------------------------------动作步骤--------------------------------------------------------
CASE station.iStepAuto OF	  
	0: //----Home Step，等待启动----
		IF station.xDisabled 
			AND station.xCanRun 
			AND NOT fbMachine[1].xStopped 
			AND NOT station.xSingleRunning 
		THEN
			station.xDone:=TRUE;
		END_IF
		
		IF  station.xSingleRunning 
			OR station.xCanRun 
			//AND NOT station.xDone 
			AND NOT station.xDisabled 
			AND NOT fbMachine[1].xStopped
		THEN
			station.xCycleEnable:=TRUE;
			//station.xDone:= FALSE;  
			
			station.iStepAuto:= 10;
		END_IF
    10: //复位数据 
			station.iStepAuto :=20;
		20://启动皮带线
			ATV12.xIMotorStart:=TRUE;
			station.iStepAuto :=999;		
		
	 999://----Single Run Finish----
		 station.iStepAuto :=0;
		 IF NOT station.xSingleContinuousRun THEN
			 station.xSingleRunFlag:=FALSE;
		 END_IF
		 
		 station.xCycleEnable:=FALSE;	
		 (*station.xDone:=TRUE;*)
	ELSE
		;	
END_CASE
END_IF
END_ACTION

